LIN {X 104.762,Y 110.384,Z 68.000,A 180.000,B 0.000,C 180.000} C_DIS
LIN {X 105.299,Y 110.068,Z 68.000,A 180.000,B 0.000,C 180.000} C_DIS
LIN {X 105.477,Y 109.954,Z 68.000,A 180.000,B 0.000,C 180.000} C_DIS
LIN {X 105.835,Y 109.715,Z 68.000,A 180.000,B 0.000,C 180.000} C_DIS
LIN {X 106.014,Y 109.595,Z 68.000,A 180.000,B 0.000,C 180.000} C_DIS
LIN {X 106.023,Y 109.589,Z 68.000,A 180.000,B 0.000,C 180.000} C_DIS
LIN {X 106.193,Y 109.465,Z 68.000,A 180.000,B 0.000,C 180.000} C_DIS
LIN {X 106.550,Y 109.196,Z 68.000,A 180.000,B 0.000,C 180.000} C_DIS
LIN {X 106.729,Y 109.060,Z 68.000,A 180.000,B 0.000,C 180.000} C_DIS
LIN {X 106.737,Y 109.053,Z 68.000,A 180.000,B 0.000,C 180.000} C_DIS
LIN {X 106.908,Y 108.910,Z 68.000,A 180.000,B 0.000,C 180.000} C_DIS
LIN {X 107.265,Y 108.608,Z 68.000,A 180.000,B 0.000,C 180.000} C_DIS
LIN {X 107.371,Y 108.517,Z 68.000,A 180.000,B 0.000,C 180.000} C_DIS
LIN {X 107.444,Y 108.448,Z 68.000,A 180.000,B 0.000,C 180.000} C_DIS
LIN {X 107.802,Y 108.110,Z 68.000,A 180.000,B 0.000,C 180.000} C_DIS
LIN {X 107.938,Y 107.980,Z 68.000,A 180.000,B 0.000,C 180.000} C_DIS
LIN {X 107.980,Y 107.938,Z 68.000,A 180.000,B 0.000,C 180.000} C_DIS
LIN {X 108.110,Y 107.802,Z 68.000,A 180.000,B 0.000,C 180.000} C_DIS
LIN {X 108.448,Y 107.444,Z 68.000,A 180.000,B 0.000,C 180.000} C_DIS
LIN {X 108.517,Y 107.371,Z 68.000,A 180.000,B 0.000,C 180.000} C_DIS
LIN {X 108.608,Y 107.265,Z 68.000,A 180.000,B 0.000,C 180.000} C_DIS
LIN {X 108.910,Y 106.908,Z 68.000,A 180.000,B 0.000,C 180.000} C_DIS
LIN {X 109.053,Y 106.737,Z 68.000,A 180.000,B 0.000,C 180.000} C_DIS
LIN {X 109.060,Y 106.729,Z 68.000,A 180.000,B 0.000,C 180.000} C_DIS
LIN {X 109.196,Y 106.550,Z 68.000,A 180.000,B 0.000,C 180.000} C_DIS
LIN {X 109.465,Y 106.193,Z 68.000,A 180.000,B 0.000,C 180.000} C_DIS
LIN {X 109.589,Y 106.023,Z 68.000,A 180.000,B 0.000,C 180.000} C_DIS
LIN {X 109.595,Y 106.014,Z 68.000,A 180.000,B 0.000,C 180.000} C_DIS
LIN {X 109.715,Y 105.835,Z 68.000,A 180.000,B 0.000,C 180.000} C_DIS
LIN {X 109.954,Y 105.477,Z 68.000,A 180.000,B 0.000,C 180.000} C_DIS
LIN {X 110.068,Y 105.299,Z 68.000,A 180.000,B 0.000,C 180.000} C_DIS
LIN {X 110.384,Y 104.762,Z 68.000,A 180.000,B 0.000,C 180.000} C_DIS
LIN {X 110.483,Y 104.586,Z 68.000,A 180.000,B 0.000,C 180.000} C_DIS
LIN {X 110.761,Y 104.047,Z 68.000,A 180.000,B 0.000,C 180.000} C_DIS
LIN {X 110.841,Y 103.889,Z 68.000,A 180.000,B 0.000,C 180.000} C_DIS
LIN {X 110.850,Y 103.869,Z 68.000,A 180.000,B 0.000,C 180.000} C_DIS
LIN {X 110.930,Y 103.690,Z 68.000,A 180.000,B 0.000,C 180.000} C_DIS
LIN {X 111.090,Y 103.332,Z 68.000,A 180.000,B 0.000,C 180.000} C_DIS
LIN {X 111.169,Y 103.153,Z 68.000,A 180.000,B 0.000,C 180.000} C_DIS
LIN {X 111.198,Y 103.079,Z 68.000,A 180.000,B 0.000,C 180.000} C_DIS
LIN {X 111.377,Y 102.610,Z 68.000,A 180.000,B 0.000,C 180.000} C_DIS
LIN {X 111.442,Y 102.438,Z 68.000,A 180.000,B 0.000,C 180.000} C_DIS
LIN {X 111.503,Y 102.260,Z 68.000,A 180.000,B 0.000,C 180.000} C_DIS
LIN {X 111.674,Y 101.723,Z 68.000,A 180.000,B 0.000,C 180.000} C_DIS
LIN {X 111.728,Y 101.545,Z 68.000,A 180.000,B 0.000,C 180.000} C_DIS
LIN {X 111.734,Y 101.518,Z 68.000,A 180.000,B 0.000,C 180.000} C_DIS
LIN {X 111.866,Y 101.008,Z 68.000,A 180.000,B 0.000,C 180.000} C_DIS
LIN {X 111.912,Y 100.829,Z 68.000,A 180.000,B 0.000,C 180.000} C_DIS
LIN {X 111.913,Y 100.824,Z 68.000,A 180.000,B 0.000,C 180.000} C_DIS
LIN {X 111.950,Y 100.651,Z 68.000,A 180.000,B 0.000,C 180.000} C_DIS
LIN {X 112.057,Y 100.114,Z 68.000,A 180.000,B 0.000,C 180.000} C_DIS
LIN {X 112.090,Y 99.936,Z 68.000,A 180.000,B 0.000,C 180.000} C_DIS
LIN {X 112.092,Y 99.919,Z 68.000,A 180.000,B 0.000,C 180.000} C_DIS
LIN {X 112.115,Y 99.757,Z 68.000,A 180.000,B 0.000,C 180.000} C_DIS
LIN {X 112.165,Y 99.399,Z 68.000,A 180.000,B 0.000,C 180.000} C_DIS
LIN {X 112.191,Y 99.221,Z 68.000,A 180.000,B 0.000,C 180.000} C_DIS
LIN {X 112.209,Y 99.042,Z 68.000,A 180.000,B 0.000,C 180.000} C_DIS
LIN {X 112.255,Y 98.505,Z 68.000,A 180.000,B 0.000,C 180.000} C_DIS
LIN {X 112.269,Y 98.327,Z 68.000,A 180.000,B 0.000,C 180.000} C_DIS
LIN {X 112.271,Y 98.281,Z 68.000,A 180.000,B 0.000,C 180.000} C_DIS
LIN {X 112.275,Y 98.148,Z 68.000,A 180.000,B 0.000,C 180.000} C_DIS
LIN {X 112.290,Y 97.612,Z 68.000,A 180.000,B 0.000,C 180.000} C_DIS
LIN {X 112.291,Y 97.433,Z 68.000,A 180.000,B 0.000,C 180.000} C_DIS
LIN {X 112.281,Y 97.075,Z 68.000,A 180.000,B 0.000,C 180.000} C_DIS
LIN {X 112.276,Y 96.897,Z 68.000,A 180.000,B 0.000,C 180.000} C_DIS
LIN {X 112.271,Y 96.719,Z 68.000,A 180.000,B 0.000,C 180.000} C_DIS
LIN {X 112.271,Y 96.718,Z 68.000,A 180.000,B 0.000,C 180.000} C_DIS
LIN {X 112.258,Y 96.539,Z 68.000,A 180.000,B 0.000,C 180.000} C_DIS
LIN {X 112.213,Y 96.003,Z 68.000,A 180.000,B 0.000,C 180.000} C_DIS
LIN {X 112.196,Y 95.824,Z 68.000,A 180.000,B 0.000,C 180.000} C_DIS
LIN {X 112.172,Y 95.645,Z 68.000,A 180.000,B 0.000,C 180.000} C_DIS
LIN {X 112.096,Y 95.109,Z 68.000,A 180.000,B 0.000,C 180.000} C_DIS
LIN {X 112.092,Y 95.081,Z 68.000,A 180.000,B 0.000,C 180.000} C_DIS
LIN {X 112.065,Y 94.930,Z 68.000,A 180.000,B 0.000,C 180.000} C_DIS
LIN {X 111.959,Y 94.394,Z 68.000,A 180.000,B 0.000,C 180.000} C_DIS
LIN {X 111.922,Y 94.215,Z 68.000,A 180.000,B 0.000,C 180.000} C_DIS
LIN {X 111.913,Y 94.176,Z 68.000,A 180.000,B 0.000,C 180.000} C_DIS
LIN {X 111.877,Y 94.036,Z 68.000,A 180.000,B 0.000,C 180.000} C_DIS
LIN {X 111.734,Y 93.482,Z 68.000,A 180.000,B 0.000,C 180.000} C_DIS
LIN {X 111.688,Y 93.321,Z 68.000,A 180.000,B 0.000,C 180.000} C_DIS
LIN {X 111.517,Y 92.785,Z 68.000,A 180.000,B 0.000,C 180.000} C_DIS
LIN {X 111.459,Y 92.606,Z 68.000,A 180.000,B 0.000,C 180.000} C_DIS
LIN {X 111.391,Y 92.427,Z 68.000,A 180.000,B 0.000,C 180.000} C_DIS
LIN {X 111.198,Y 91.921,Z 68.000,A 180.000,B 0.000,C 180.000} C_DIS
LIN {X 111.186,Y 91.891,Z 68.000,A 180.000,B 0.000,C 180.000} C_DIS
LIN {X 111.110,Y 91.712,Z 68.000,A 180.000,B 0.000,C 180.000} C_DIS
LIN {X 110.870,Y 91.176,Z 68.000,A 180.000,B 0.000,C 180.000} C_DIS
LIN {X 110.841,Y 91.111,Z 68.000,A 180.000,B 0.000,C 180.000} C_DIS
LIN {X 110.784,Y 90.997,Z 68.000,A 180.000,B 0.000,C 180.000} C_DIS
LIN {X 110.483,Y 90.414,Z 68.000,A 180.000,B 0.000,C 180.000} C_DIS
LIN {X 110.410,Y 90.282,Z 68.000,A 180.000,B 0.000,C 180.000} C_DIS
LIN {X 110.113,Y 89.778,Z 68.000,A 180.000,B 0.000,C 180.000} C_DIS
; Link Move Starts
LIN {X 109.952,Y 89.519,Z 68.000,A 180.000,B 0.000,C 180.000} C_DIS
LIN {X 109.779,Y 89.258,Z 67.999,A 180.000,B 0.000,C 180.000} C_DIS
LIN {X 109.604,Y 88.996,Z 67.998,A 180.000,B 0.000,C 180.000} C_DIS
LIN {X 109.425,Y 88.751,Z 67.996,A 180.000,B 0.000,C 180.000} C_DIS
LIN {X 109.237,Y 88.499,Z 67.994,A 180.000,B 0.000,C 180.000} C_DIS
LIN {X 109.053,Y 88.256,Z 67.992,A 180.000,B 0.000,C 180.000} C_DIS
LIN {X 108.852,Y 88.015,Z 67.989,A 180.000,B 0.000,C 180.000} C_DIS
LIN {X 108.650,Y 87.773,Z 67.985,A 180.000,B 0.000,C 180.000} C_DIS
LIN {X 108.450,Y 87.544,Z 67.982,A 180.000,B 0.000,C 180.000} C_DIS
LIN {X 108.235,Y 87.314,Z 67.977,A 180.000,B 0.000,C 180.000} C_DIS
LIN {X 108.020,Y 87.084,Z 67.973,A 180.000,B 0.000,C 180.000} C_DIS
LIN {X 107.803,Y 86.870,Z 67.968,A 180.000,B 0.000,C 180.000} C_DIS
LIN {X 107.690,Y 86.761,Z 67.965,A 180.000,B 0.000,C 180.000} C_DIS
LIN {X 107.576,Y 86.652,Z 67.962,A 180.000,B 0.000,C 180.000} C_DIS
LIN {X 107.465,Y 86.545,Z 67.960,A 180.000,B 0.000,C 180.000} C_DIS
LIN {X 107.352,Y 86.439,Z 67.957,A 180.000,B 0.000,C 180.000} C_DIS
LIN {X 107.235,Y 86.338,Z 67.954,A 180.000,B 0.000,C 180.000} C_DIS
LIN {X 107.117,Y 86.236,Z 67.951,A 180.000,B 0.000,C 180.000} C_DIS
LIN {X 106.998,Y 86.134,Z 67.947,A 180.000,B 0.000,C 180.000} C_DIS
LIN {X 106.878,Y 86.031,Z 67.944,A 180.000,B 0.000,C 180.000} C_DIS
LIN {X 106.762,Y 85.931,Z 67.941,A 180.000,B 0.000,C 180.000} C_DIS
LIN {X 106.641,Y 85.835,Z 67.937,A 180.000,B 0.000,C 180.000} C_DIS
LIN {X 106.517,Y 85.740,Z 67.934,A 180.000,B 0.000,C 180.000} C_DIS
LIN {X 106.393,Y 85.645,Z 67.930,A 180.000,B 0.000,C 180.000} C_DIS
LIN {X 106.269,Y 85.549,Z 67.926,A 180.000,B 0.000,C 180.000} C_DIS
LIN {X 106.144,Y 85.453,Z 67.923,A 180.000,B 0.000,C 180.000} C_DIS
LIN {X 106.021,Y 85.363,Z 67.919,A 180.000,B 0.000,C 180.000} C_DIS
LIN {X 105.894,Y 85.276,Z 67.915,A 180.000,B 0.000,C 180.000} C_DIS
LIN {X 105.765,Y 85.187,Z 67.911,A 180.000,B 0.000,C 180.000} C_DIS
LIN {X 105.635,Y 85.098,Z 67.907,A 180.000,B 0.000,C 180.000} C_DIS
LIN {X 105.508,Y 85.011,Z 67.903,A 180.000,B 0.000,C 180.000} C_DIS
LIN {X 105.380,Y 84.926,Z 67.899,A 180.000,B 0.000,C 180.000} C_DIS
LIN {X 105.247,Y 84.844,Z 67.894,A 180.000,B 0.000,C 180.000} C_DIS
LIN {X 105.113,Y 84.762,Z 67.890,A 180.000,B 0.000,C 180.000} C_DIS
LIN {X 104.978,Y 84.680,Z 67.885,A 180.000,B 0.000,C 180.000} C_DIS
LIN {X 104.844,Y 84.599,Z 67.881,A 180.000,B 0.000,C 180.000} C_DIS
LIN {X 104.712,Y 84.519,Z 67.876,A 180.000,B 0.000,C 180.000} C_DIS
LIN {X 104.577,Y 84.444,Z 67.872,A 180.000,B 0.000,C 180.000} C_DIS
LIN {X 104.439,Y 84.370,Z 67.867,A 180.000,B 0.000,C 180.000} C_DIS
LIN {X 104.300,Y 84.296,Z 67.862,A 180.000,B 0.000,C 180.000} C_DIS
LIN {X 104.162,Y 84.222,Z 67.857,A 180.000,B 0.000,C 180.000} C_DIS
LIN {X 104.023,Y 84.148,Z 67.852,A 180.000,B 0.000,C 180.000} C_DIS
LIN {X 103.885,Y 84.079,Z 67.847,A 180.000,B 0.000,C 180.000} C_DIS
LIN {X 103.746,Y 84.014,Z 67.842,A 180.000,B 0.000,C 180.000} C_DIS
LIN {X 103.675,Y 83.981,Z 67.840,A 180.000,B 0.000,C 180.000} C_DIS
LIN {X 103.603,Y 83.947,Z 67.837,A 180.000,B 0.000,C 180.000} C_DIS
LIN {X 103.532,Y 83.914,Z 67.835,A 180.000,B 0.000,C 180.000} C_DIS
LIN {X 103.390,Y 83.848,Z 67.829,A 180.000,B 0.000,C 180.000} C_DIS
LIN {X 103.319,Y 83.815,Z 67.827,A 180.000,B 0.000,C 180.000} C_DIS
LIN {X 103.249,Y 83.782,Z 67.824,A 180.000,B 0.000,C 180.000} C_DIS
LIN {X 103.178,Y 83.751,Z 67.821,A 180.000,B 0.000,C 180.000} C_DIS
LIN {X 103.106,Y 83.721,Z 67.819,A 180.000,B 0.000,C 180.000} C_DIS
LIN {X 103.033,Y 83.692,Z 67.816,A 180.000,B 0.000,C 180.000} C_DIS
LIN {X 102.888,Y 83.634,Z 67.811,A 180.000,B 0.000,C 180.000} C_DIS
LIN {X 102.742,Y 83.576,Z 67.805,A 180.000,B 0.000,C 180.000} C_DIS
LIN {X 102.524,Y 83.488,Z 67.797,A 180.000,B 0.000,C 180.000} C_DIS
LIN {X 102.453,Y 83.460,Z 67.794,A 180.000,B 0.000,C 180.000} C_DIS
LIN {X 102.380,Y 83.433,Z 67.792,A 180.000,B 0.000,C 180.000} C_DIS
LIN {X 102.307,Y 83.408,Z 67.789,A 180.000,B 0.000,C 180.000} C_DIS
LIN {X 102.158,Y 83.358,Z 67.783,A 180.000,B 0.000,C 180.000} C_DIS
LIN {X 101.934,Y 83.283,Z 67.775,A 180.000,B 0.000,C 180.000} C_DIS
LIN {X 101.784,Y 83.232,Z 67.770,A 180.000,B 0.000,C 180.000} C_DIS
LIN {X 101.710,Y 83.207,Z 67.767,A 180.000,B 0.000,C 180.000} C_DIS
LIN {X 101.636,Y 83.183,Z 67.764,A 180.000,B 0.000,C 180.000} C_DIS
LIN {X 101.562,Y 83.161,Z 67.762,A 180.000,B 0.000,C 180.000} C_DIS
LIN {X 101.413,Y 83.120,Z 67.756,A 180.000,B 0.000,C 180.000} C_DIS
LIN {X 101.261,Y 83.078,Z 67.751,A 180.000,B 0.000,C 180.000} C_DIS
LIN {X 101.034,Y 83.016,Z 67.742,A 180.000,B 0.000,C 180.000} C_DIS
LIN {X 100.884,Y 82.975,Z 67.737,A 180.000,B 0.000,C 180.000} C_DIS
LIN {X 100.809,Y 82.955,Z 67.734,A 180.000,B 0.000,C 180.000} C_DIS
LIN {X 100.732,Y 82.938,Z 67.732,A 180.000,B 0.000,C 180.000} C_DIS
LIN {X 100.578,Y 82.905,Z 67.726,A 180.000,B 0.000,C 180.000} C_DIS
LIN {X 100.502,Y 82.888,Z 67.723,A 180.000,B 0.000,C 180.000} C_DIS
LIN {X 100.348,Y 82.855,Z 67.718,A 180.000,B 0.000,C 180.000} C_DIS
LIN {X 100.118,Y 82.805,Z 67.710,A 180.000,B 0.000,C 180.000} C_DIS
LIN {X 100.042,Y 82.789,Z 67.707,A 180.000,B 0.000,C 180.000} C_DIS
LIN {X 99.965,Y 82.775,Z 67.704,A 180.000,B 0.000,C 180.000} C_DIS
LIN {X 99.888,Y 82.762,Z 67.701,A 180.000,B 0.000,C 180.000} C_DIS
LIN {X 99.733,Y 82.738,Z 67.696,A 180.000,B 0.000,C 180.000} C_DIS
LIN {X 99.266,Y 82.664,Z 67.679,A 180.000,B 0.000,C 180.000} C_DIS
LIN {X 99.189,Y 82.653,Z 67.677,A 180.000,B 0.000,C 180.000} C_DIS
LIN {X 99.112,Y 82.643,Z 67.674,A 180.000,B 0.000,C 180.000} C_DIS
LIN {X 98.956,Y 82.628,Z 67.669,A 180.000,B 0.000,C 180.000} C_DIS
LIN {X 98.800,Y 82.612,Z 67.663,A 180.000,B 0.000,C 180.000} C_DIS
LIN {X 98.408,Y 82.572,Z 67.649,A 180.000,B 0.000,C 180.000} C_DIS
LIN {X 98.330,Y 82.566,Z 67.647,A 180.000,B 0.000,C 180.000} C_DIS
LIN {X 98.252,Y 82.562,Z 67.644,A 180.000,B 0.000,C 180.000} C_DIS
LIN {X 97.781,Y 82.541,Z 67.627,A 180.000,B 0.000,C 180.000} C_DIS
LIN {X 97.624,Y 82.534,Z 67.622,A 180.000,B 0.000,C 180.000} C_DIS
LIN {X 97.546,Y 82.530,Z 67.619,A 180.000,B 0.000,C 180.000} C_DIS
LIN {X 97.467,Y 82.529,Z 67.616,A 180.000,B 0.000,C 180.000} C_DIS
LIN {X 97.389,Y 82.530,Z 67.614,A 180.000,B 0.000,C 180.000} C_DIS
LIN {X 97.153,Y 82.532,Z 67.605,A 180.000,B 0.000,C 180.000} C_DIS
LIN {X 96.995,Y 82.534,Z 67.600,A 180.000,B 0.000,C 180.000} C_DIS
LIN {X 96.759,Y 82.537,Z 67.592,A 180.000,B 0.000,C 180.000} C_DIS
LIN {X 96.680,Y 82.538,Z 67.589,A 180.000,B 0.000,C 180.000} C_DIS
LIN {X 96.602,Y 82.542,Z 67.586,A 180.000,B 0.000,C 180.000} C_DIS
LIN {X 96.524,Y 82.547,Z 67.583,A 180.000,B 0.000,C 180.000} C_DIS
LIN {X 96.131,Y 82.574,Z 67.570,A 180.000,B 0.000,C 180.000} C_DIS
LIN {X 95.895,Y 82.590,Z 67.561,A 180.000,B 0.000,C 180.000} C_DIS
LIN {X 95.817,Y 82.597,Z 67.559,A 180.000,B 0.000,C 180.000} C_DIS
LIN {X 95.739,Y 82.605,Z 67.556,A 180.000,B 0.000,C 180.000} C_DIS
LIN {X 95.709,Y 82.609,Z 67.555,A 180.000,B 0.000,C 180.000} C_DIS
LIN {X 95.115,Y 82.693,Z 67.534,A 180.000,B 0.000,C 180.000} C_DIS
LIN {X 95.037,Y 82.704,Z 67.531,A 180.000,B 0.000,C 180.000} C_DIS
LIN {X 94.959,Y 82.717,Z 67.528,A 180.000,B 0.000,C 180.000} C_DIS
LIN {X 94.882,Y 82.732,Z 67.526,A 180.000,B 0.000,C 180.000} C_DIS
LIN {X 94.264,Y 82.855,Z 67.504,A 180.000,B 0.000,C 180.000} C_DIS
LIN {X 94.187,Y 82.871,Z 67.501,A 180.000,B 0.000,C 180.000} C_DIS
LIN {X 94.110,Y 82.889,Z 67.498,A 180.000,B 0.000,C 180.000} C_DIS
LIN {X 94.034,Y 82.908,Z 67.495,A 180.000,B 0.000,C 180.000} C_DIS
LIN {X 93.424,Y 83.066,Z 67.473,A 180.000,B 0.000,C 180.000} C_DIS
LIN {X 93.348,Y 83.086,Z 67.471,A 180.000,B 0.000,C 180.000} C_DIS
LIN {X 93.272,Y 83.109,Z 67.468,A 180.000,B 0.000,C 180.000} C_DIS
LIN {X 92.672,Y 83.300,Z 67.446,A 180.000,B 0.000,C 180.000} C_DIS
LIN {X 92.597,Y 83.324,Z 67.443,A 180.000,B 0.000,C 180.000} C_DIS
LIN {X 92.523,Y 83.350,Z 67.440,A 180.000,B 0.000,C 180.000} C_DIS
LIN {X 92.449,Y 83.378,Z 67.438,A 180.000,B 0.000,C 180.000} C_DIS
LIN {X 92.007,Y 83.546,Z 67.421,A 180.000,B 0.000,C 180.000} C_DIS
LIN {X 91.860,Y 83.602,Z 67.416,A 180.000,B 0.000,C 180.000} C_DIS
LIN {X 91.787,Y 83.631,Z 67.413,A 180.000,B 0.000,C 180.000} C_DIS
LIN {X 91.714,Y 83.661,Z 67.410,A 180.000,B 0.000,C 180.000} C_DIS
LIN {X 91.642,Y 83.693,Z 67.407,A 180.000,B 0.000,C 180.000} C_DIS
LIN {X 91.427,Y 83.790,Z 67.399,A 180.000,B 0.000,C 180.000} C_DIS
LIN {X 91.067,Y 83.951,Z 67.385,A 180.000,B 0.000,C 180.000} C_DIS
LIN {X 90.996,Y 83.984,Z 67.383,A 180.000,B 0.000,C 180.000} C_DIS
LIN {X 90.925,Y 84.019,Z 67.380,A 180.000,B 0.000,C 180.000} C_DIS
LIN {X 90.505,Y 84.236,Z 67.363,A 180.000,B 0.000,C 180.000} C_DIS
LIN {X 90.365,Y 84.308,Z 67.358,A 180.000,B 0.000,C 180.000} C_DIS
LIN {X 90.296,Y 84.344,Z 67.355,A 180.000,B 0.000,C 180.000} C_DIS
LIN {X 90.226,Y 84.382,Z 67.352,A 180.000,B 0.000,C 180.000} C_DIS
LIN {X 90.158,Y 84.421,Z 67.350,A 180.000,B 0.000,C 180.000} C_DIS
LIN {X 89.955,Y 84.541,Z 67.341,A 180.000,B 0.000,C 180.000} C_DIS
LIN {X 89.819,Y 84.621,Z 67.336,A 180.000,B 0.000,C 180.000} C_DIS
LIN {X 89.683,Y 84.701,Z 67.330,A 180.000,B 0.000,C 180.000} C_DIS
LIN {X 89.616,Y 84.741,Z 67.328,A 180.000,B 0.000,C 180.000} C_DIS
LIN {X 89.548,Y 84.782,Z 67.325,A 180.000,B 0.000,C 180.000} C_DIS
LIN {X 89.481,Y 84.824,Z 67.322,A 180.000,B 0.000,C 180.000} C_DIS
LIN {X 89.416,Y 84.867,Z 67.319,A 180.000,B 0.000,C 180.000} C_DIS
LIN {X 89.350,Y 84.911,Z 67.317,A 180.000,B 0.000,C 180.000} C_DIS
LIN {X 89.219,Y 84.999,Z 67.311,A 180.000,B 0.000,C 180.000} C_DIS
LIN {X 88.892,Y 85.217,Z 67.297,A 180.000,B 0.000,C 180.000} C_DIS
LIN {X 88.827,Y 85.262,Z 67.295,A 180.000,B 0.000,C 180.000} C_DIS
LIN {X 88.763,Y 85.308,Z 67.292,A 180.000,B 0.000,C 180.000} C_DIS
LIN {X 88.637,Y 85.403,Z 67.286,A 180.000,B 0.000,C 180.000} C_DIS
LIN {X 88.574,Y 85.450,Z 67.284,A 180.000,B 0.000,C 180.000} C_DIS
LIN {X 88.449,Y 85.545,Z 67.278,A 180.000,B 0.000,C 180.000} C_DIS
LIN {X 88.260,Y 85.687,Z 67.270,A 180.000,B 0.000,C 180.000} C_DIS
LIN {X 88.197,Y 85.734,Z 67.267,A 180.000,B 0.000,C 180.000} C_DIS
LIN {X 88.135,Y 85.783,Z 67.265,A 180.000,B 0.000,C 180.000} C_DIS
LIN {X 88.074,Y 85.833,Z 67.262,A 180.000,B 0.000,C 180.000} C_DIS
LIN {X 87.954,Y 85.935,Z 67.256,A 180.000,B 0.000,C 180.000} C_DIS
LIN {X 87.774,Y 86.087,Z 67.248,A 180.000,B 0.000,C 180.000} C_DIS
LIN {X 87.653,Y 86.189,Z 67.243,A 180.000,B 0.000,C 180.000} C_DIS
LIN {X 87.593,Y 86.240,Z 67.240,A 180.000,B 0.000,C 180.000} C_DIS
LIN {X 87.533,Y 86.291,Z 67.237,A 180.000,B 0.000,C 180.000} C_DIS
LIN {X 87.474,Y 86.343,Z 67.234,A 180.000,B 0.000,C 180.000} C_DIS
LIN {X 87.417,Y 86.397,Z 67.232,A 180.000,B 0.000,C 180.000} C_DIS
LIN {X 87.360,Y 86.451,Z 67.229,A 180.000,B 0.000,C 180.000} C_DIS
LIN {X 87.245,Y 86.559,Z 67.223,A 180.000,B 0.000,C 180.000} C_DIS
LIN {X 87.074,Y 86.722,Z 67.215,A 180.000,B 0.000,C 180.000} C_DIS
LIN {X 86.959,Y 86.830,Z 67.210,A 180.000,B 0.000,C 180.000} C_DIS
LIN {X 86.902,Y 86.884,Z 67.207,A 180.000,B 0.000,C 180.000} C_DIS
LIN {X 86.847,Y 86.941,Z 67.204,A 180.000,B 0.000,C 180.000} C_DIS
LIN {X 86.739,Y 87.055,Z 67.199,A 180.000,B 0.000,C 180.000} C_DIS
LIN {X 86.685,Y 87.112,Z 67.196,A 180.000,B 0.000,C 180.000} C_DIS
LIN {X 86.577,Y 87.227,Z 67.190,A 180.000,B 0.000,C 180.000} C_DIS
LIN {X 86.469,Y 87.341,Z 67.185,A 180.000,B 0.000,C 180.000} C_DIS
LIN {X 86.360,Y 87.456,Z 67.179,A 180.000,B 0.000,C 180.000} C_DIS
LIN {X 86.307,Y 87.514,Z 67.177,A 180.000,B 0.000,C 180.000} C_DIS
LIN {X 86.256,Y 87.574,Z 67.174,A 180.000,B 0.000,C 180.000} C_DIS
LIN {X 86.154,Y 87.694,Z 67.169,A 180.000,B 0.000,C 180.000} C_DIS
LIN {X 86.053,Y 87.814,Z 67.164,A 180.000,B 0.000,C 180.000} C_DIS
LIN {X 86.002,Y 87.874,Z 67.161,A 180.000,B 0.000,C 180.000} C_DIS
LIN {X 85.951,Y 87.935,Z 67.158,A 180.000,B 0.000,C 180.000} C_DIS
LIN {X 85.900,Y 87.995,Z 67.156,A 180.000,B 0.000,C 180.000} C_DIS
LIN {X 85.850,Y 88.055,Z 67.153,A 180.000,B 0.000,C 180.000} C_DIS
LIN {X 85.799,Y 88.115,Z 67.151,A 180.000,B 0.000,C 180.000} C_DIS
LIN {X 85.750,Y 88.177,Z 67.148,A 180.000,B 0.000,C 180.000} C_DIS
LIN {X 85.655,Y 88.302,Z 67.143,A 180.000,B 0.000,C 180.000} C_DIS
LIN {X 85.560,Y 88.428,Z 67.138,A 180.000,B 0.000,C 180.000} C_DIS
LIN {X 85.465,Y 88.554,Z 67.134,A 180.000,B 0.000,C 180.000} C_DIS
LIN {X 85.371,Y 88.680,Z 67.129,A 180.000,B 0.000,C 180.000} C_DIS
LIN {X 85.276,Y 88.806,Z 67.124,A 180.000,B 0.000,C 180.000} C_DIS
LIN {X 85.188,Y 88.936,Z 67.120,A 180.000,B 0.000,C 180.000} C_DIS
LIN {X 85.100,Y 89.067,Z 67.115,A 180.000,B 0.000,C 180.000} C_DIS
LIN {X 85.013,Y 89.198,Z 67.110,A 180.000,B 0.000,C 180.000} C_DIS
LIN {X 84.925,Y 89.329,Z 67.106,A 180.000,B 0.000,C 180.000} C_DIS
LIN {X 84.838,Y 89.460,Z 67.102,A 180.000,B 0.000,C 180.000} C_DIS
LIN {X 84.754,Y 89.594,Z 67.097,A 180.000,B 0.000,C 180.000} C_DIS
LIN {X 84.674,Y 89.729,Z 67.093,A 180.000,B 0.000,C 180.000} C_DIS
LIN {X 84.594,Y 89.865,Z 67.089,A 180.000,B 0.000,C 180.000} C_DIS
LIN {X 84.514,Y 90.001,Z 67.085,A 180.000,B 0.000,C 180.000} C_DIS
LIN {X 84.434,Y 90.136,Z 67.081,A 180.000,B 0.000,C 180.000} C_DIS
LIN {X 84.356,Y 90.273,Z 67.077,A 180.000,B 0.000,C 180.000} C_DIS
LIN {X 84.283,Y 90.413,Z 67.073,A 180.000,B 0.000,C 180.000} C_DIS
LIN {X 84.211,Y 90.553,Z 67.070,A 180.000,B 0.000,C 180.000} C_DIS
LIN {X 84.139,Y 90.693,Z 67.066,A 180.000,B 0.000,C 180.000} C_DIS
LIN {X 84.067,Y 90.833,Z 67.062,A 180.000,B 0.000,C 180.000} C_DIS
LIN {X 83.995,Y 90.973,Z 67.059,A 180.000,B 0.000,C 180.000} C_DIS
LIN {X 83.929,Y 91.116,Z 67.056,A 180.000,B 0.000,C 180.000} C_DIS
LIN {X 83.865,Y 91.260,Z 67.052,A 180.000,B 0.000,C 180.000} C_DIS
LIN {X 83.800,Y 91.403,Z 67.049,A 180.000,B 0.000,C 180.000} C_DIS
LIN {X 83.736,Y 91.547,Z 67.046,A 180.000,B 0.000,C 180.000} C_DIS
LIN {X 83.672,Y 91.691,Z 67.043,A 180.000,B 0.000,C 180.000} C_DIS
LIN {X 83.611,Y 91.837,Z 67.040,A 180.000,B 0.000,C 180.000} C_DIS
LIN {X 83.555,Y 91.984,Z 67.037,A 180.000,B 0.000,C 180.000} C_DIS
LIN {X 83.499,Y 92.131,Z 67.034,A 180.000,B 0.000,C 180.000} C_DIS
LIN {X 83.443,Y 92.278,Z 67.032,A 180.000,B 0.000,C 180.000} C_DIS
LIN {X 83.387,Y 92.425,Z 67.029,A 180.000,B 0.000,C 180.000} C_DIS
LIN {X 83.284,Y 92.723,Z 67.024,A 180.000,B 0.000,C 180.000} C_DIS
LIN {X 83.189,Y 93.023,Z 67.020,A 180.000,B 0.000,C 180.000} C_DIS
LIN {X 83.093,Y 93.323,Z 67.016,A 180.000,B 0.000,C 180.000} C_DIS
LIN {X 83.013,Y 93.628,Z 67.013,A 180.000,B 0.000,C 180.000} C_DIS
LIN {X 82.934,Y 93.933,Z 67.009,A 180.000,B 0.000,C 180.000} C_DIS
LIN {X 82.860,Y 94.239,Z 67.007,A 180.000,B 0.000,C 180.000} C_DIS
LIN {X 82.798,Y 94.548,Z 67.004,A 180.000,B 0.000,C 180.000} C_DIS
LIN {X 82.737,Y 94.857,Z 67.003,A 180.000,B 0.000,C 180.000} C_DIS
LIN {X 82.686,Y 95.167,Z 67.001,A 180.000,B 0.000,C 180.000} C_DIS
LIN {X 82.641,Y 95.479,Z 67.000,A 180.000,B 0.000,C 180.000} C_DIS
LIN {X 82.598,Y 95.791,Z 67.000,A 180.000,B 0.000,C 180.000} C_DIS
LIN {X 82.589,Y 95.875,Z 67.000,A 180.000,B 0.000,C 180.000} C_DIS
; Cutting Move Starts
LIN {X 82.578,Y 96.003,Z 67.000,A 180.000,B 0.000,C 180.000} C_DIS
LIN {X 82.533,Y 96.539,Z 67.000,A 180.000,B 0.000,C 180.000} C_DIS
LIN {X 82.521,Y 96.718,Z 67.000,A 180.000,B 0.000,C 180.000} C_DIS
LIN {X 82.516,Y 96.897,Z 67.000,A 180.000,B 0.000,C 180.000} C_DIS
LIN {X 82.501,Y 97.433,Z 67.000,A 180.000,B 0.000,C 180.000} C_DIS
LIN {X 82.502,Y 97.612,Z 67.000,A 180.000,B 0.000,C 180.000} C_DIS
LIN {X 82.517,Y 98.148,Z 67.000,A 180.000,B 0.000,C 180.000} C_DIS
LIN {X 82.523,Y 98.327,Z 67.000,A 180.000,B 0.000,C 180.000} C_DIS
LIN {X 82.536,Y 98.505,Z 67.000,A 180.000,B 0.000,C 180.000} C_DIS
LIN {X 82.582,Y 99.042,Z 67.000,A 180.000,B 0.000,C 180.000} C_DIS
LIN {X 82.595,Y 99.185,Z 67.000,A 180.000,B 0.000,C 180.000} C_DIS
LIN {X 82.599,Y 99.221,Z 67.000,A 180.000,B 0.000,C 180.000} C_DIS
LIN {X 82.624,Y 99.399,Z 67.000,A 180.000,B 0.000,C 180.000} C_DIS
LIN {X 82.700,Y 99.936,Z 67.000,A 180.000,B 0.000,C 180.000} C_DIS
LIN {X 82.731,Y 100.114,Z 67.000,A 180.000,B 0.000,C 180.000} C_DIS
LIN {X 82.838,Y 100.651,Z 67.000,A 180.000,B 0.000,C 180.000} C_DIS
LIN {X 82.874,Y 100.829,Z 67.000,A 180.000,B 0.000,C 180.000} C_DIS
LIN {X 82.919,Y 101.008,Z 67.000,A 180.000,B 0.000,C 180.000} C_DIS
LIN {X 83.057,Y 101.545,Z 67.000,A 180.000,B 0.000,C 180.000} C_DIS
LIN {X 83.108,Y 101.723,Z 67.000,A 180.000,B 0.000,C 180.000} C_DIS
LIN {X 83.310,Y 102.358,Z 67.000,A 180.000,B 0.000,C 180.000} C_DIS
LIN {X 83.336,Y 102.438,Z 67.000,A 180.000,B 0.000,C 180.000} C_DIS
LIN {X 83.403,Y 102.617,Z 67.000,A 180.000,B 0.000,C 180.000} C_DIS
LIN {X 83.608,Y 103.153,Z 67.000,A 180.000,B 0.000,C 180.000} C_DIS
LIN {X 83.668,Y 103.300,Z 67.000,A 180.000,B 0.000,C 180.000} C_DIS
LIN {X 83.922,Y 103.869,Z 67.000,A 180.000,B 0.000,C 180.000} C_DIS
LIN {X 84.005,Y 104.047,Z 67.000,A 180.000,B 0.000,C 180.000} C_DIS
LIN {X 84.025,Y 104.087,Z 67.000,A 180.000,B 0.000,C 180.000} C_DIS
LIN {X 84.282,Y 104.584,Z 67.000,A 180.000,B 0.000,C 180.000} C_DIS
LIN {X 84.375,Y 104.762,Z 67.000,A 180.000,B 0.000,C 180.000} C_DIS
LIN {X 84.383,Y 104.775,Z 67.000,A 180.000,B 0.000,C 180.000} C_DIS
LIN {X 84.480,Y 104.941,Z 67.000,A 180.000,B 0.000,C 180.000} C_DIS
LIN {X 84.740,Y 105.382,Z 67.000,A 180.000,B 0.000,C 180.000} C_DIS
LIN {X 84.797,Y 105.477,Z 67.000,A 180.000,B 0.000,C 180.000} C_DIS
LIN {X 84.915,Y 105.656,Z 67.000,A 180.000,B 0.000,C 180.000} C_DIS
LIN {X 85.154,Y 106.014,Z 67.000,A 180.000,B 0.000,C 180.000} C_DIS
LIN {X 85.276,Y 106.193,Z 67.000,A 180.000,B 0.000,C 180.000} C_DIS
LIN {X 85.276,Y 106.194,Z 67.000,A 180.000,B 0.000,C 180.000} C_DIS
LIN {X 85.409,Y 106.371,Z 67.000,A 180.000,B 0.000,C 180.000} C_DIS
LIN {X 85.678,Y 106.729,Z 67.000,A 180.000,B 0.000,C 180.000} C_DIS
LIN {X 85.813,Y 106.902,Z 67.000,A 180.000,B 0.000,C 180.000} C_DIS
LIN {X 85.818,Y 106.908,Z 67.000,A 180.000,B 0.000,C 180.000} C_DIS
LIN {X 86.271,Y 107.444,Z 67.000,A 180.000,B 0.000,C 180.000} C_DIS
LIN {X 86.349,Y 107.532,Z 67.000,A 180.000,B 0.000,C 180.000} C_DIS
LIN {X 86.435,Y 107.623,Z 67.000,A 180.000,B 0.000,C 180.000} C_DIS
LIN {X 86.773,Y 107.980,Z 67.000,A 180.000,B 0.000,C 180.000} C_DIS
LIN {X 86.885,Y 108.099,Z 67.000,A 180.000,B 0.000,C 180.000} C_DIS
LIN {X 86.947,Y 108.159,Z 67.000,A 180.000,B 0.000,C 180.000} C_DIS
LIN {X 87.422,Y 108.607,Z 67.000,A 180.000,B 0.000,C 180.000} C_DIS
LIN {X 87.517,Y 108.695,Z 67.000,A 180.000,B 0.000,C 180.000} C_DIS
LIN {X 87.601,Y 108.767,Z 67.000,A 180.000,B 0.000,C 180.000} C_DIS
LIN {X 87.958,Y 109.069,Z 67.000,A 180.000,B 0.000,C 180.000} C_DIS
LIN {X 88.137,Y 109.219,Z 67.000,A 180.000,B 0.000,C 180.000} C_DIS
LIN {X 88.153,Y 109.232,Z 67.000,A 180.000,B 0.000,C 180.000} C_DIS
LIN {X 88.316,Y 109.355,Z 67.000,A 180.000,B 0.000,C 180.000} C_DIS
LIN {X 88.673,Y 109.624,Z 67.000,A 180.000,B 0.000,C 180.000} C_DIS
LIN {X 88.852,Y 109.756,Z 67.000,A 180.000,B 0.000,C 180.000} C_DIS
LIN {X 88.870,Y 109.768,Z 67.000,A 180.000,B 0.000,C 180.000} C_DIS
LIN {X 89.031,Y 109.875,Z 67.000,A 180.000,B 0.000,C 180.000} C_DIS
LIN {X 89.405,Y 110.126,Z 67.000,A 180.000,B 0.000,C 180.000} C_DIS
LIN {X 89.567,Y 110.230,Z 67.000,A 180.000,B 0.000,C 180.000} C_DIS
LIN {X 89.693,Y 110.304,Z 67.000,A 180.000,B 0.000,C 180.000} C_DIS
LIN {X 90.103,Y 110.546,Z 67.000,A 180.000,B 0.000,C 180.000} C_DIS
LIN {X 90.282,Y 110.649,Z 67.000,A 180.000,B 0.000,C 180.000} C_DIS
LIN {X 90.307,Y 110.662,Z 67.000,A 180.000,B 0.000,C 180.000} C_DIS
LIN {X 90.818,Y 110.926,Z 67.000,A 180.000,B 0.000,C 180.000} C_DIS
LIN {X 90.997,Y 111.017,Z 67.000,A 180.000,B 0.000,C 180.000} C_DIS
LIN {X 91.002,Y 111.019,Z 67.000,A 180.000,B 0.000,C 180.000} C_DIS
LIN {X 91.176,Y 111.098,Z 67.000,A 180.000,B 0.000,C 180.000} C_DIS
LIN {X 91.533,Y 111.258,Z 67.000,A 180.000,B 0.000,C 180.000} C_DIS
LIN {X 91.712,Y 111.338,Z 67.000,A 180.000,B 0.000,C 180.000} C_DIS
LIN {X 91.806,Y 111.377,Z 67.000,A 180.000,B 0.000,C 180.000} C_DIS
LIN {X 91.891,Y 111.409,Z 67.000,A 180.000,B 0.000,C 180.000} C_DIS
LIN {X 92.427,Y 111.614,Z 67.000,A 180.000,B 0.000,C 180.000} C_DIS
LIN {X 92.606,Y 111.678,Z 67.000,A 180.000,B 0.000,C 180.000} C_DIS
LIN {X 92.964,Y 111.792,Z 67.000,A 180.000,B 0.000,C 180.000} C_DIS
LIN {X 93.142,Y 111.849,Z 67.000,A 180.000,B 0.000,C 180.000} C_DIS
LIN {X 93.321,Y 111.906,Z 67.000,A 180.000,B 0.000,C 180.000} C_DIS
LIN {X 93.346,Y 111.913,Z 67.000,A 180.000,B 0.000,C 180.000} C_DIS
LIN {X 93.500,Y 111.954,Z 67.000,A 180.000,B 0.000,C 180.000} C_DIS
LIN {X 94.036,Y 112.092,Z 67.000,A 180.000,B 0.000,C 180.000} C_DIS
LIN {X 94.215,Y 112.135,Z 67.000,A 180.000,B 0.000,C 180.000} C_DIS
LIN {X 94.394,Y 112.171,Z 67.000,A 180.000,B 0.000,C 180.000} C_DIS
LIN {X 94.895,Y 112.271,Z 67.000,A 180.000,B 0.000,C 180.000} C_DIS
LIN {X 94.930,Y 112.278,Z 67.000,A 180.000,B 0.000,C 180.000} C_DIS
LIN {X 95.109,Y 112.306,Z 67.000,A 180.000,B 0.000,C 180.000} C_DIS
LIN {X 95.645,Y 112.382,Z 67.000,A 180.000,B 0.000,C 180.000} C_DIS
LIN {X 95.824,Y 112.406,Z 67.000,A 180.000,B 0.000,C 180.000} C_DIS
LIN {X 96.003,Y 112.422,Z 67.000,A 180.000,B 0.000,C 180.000} C_DIS
LIN {X 96.539,Y 112.467,Z 67.000,A 180.000,B 0.000,C 180.000} C_DIS
LIN {X 96.718,Y 112.479,Z 67.000,A 180.000,B 0.000,C 180.000} C_DIS
LIN {X 96.897,Y 112.484,Z 67.000,A 180.000,B 0.000,C 180.000} C_DIS
LIN {X 97.433,Y 112.499,Z 67.000,A 180.000,B 0.000,C 180.000} C_DIS
LIN {X 97.612,Y 112.498,Z 67.000,A 180.000,B 0.000,C 180.000} C_DIS
LIN {X 98.148,Y 112.483,Z 67.000,A 180.000,B 0.000,C 180.000} C_DIS
LIN {X 98.327,Y 112.477,Z 67.000,A 180.000,B 0.000,C 180.000} C_DIS
LIN {X 98.505,Y 112.464,Z 67.000,A 180.000,B 0.000,C 180.000} C_DIS
LIN {X 99.042,Y 112.418,Z 67.000,A 180.000,B 0.000,C 180.000} C_DIS
LIN {X 99.221,Y 112.401,Z 67.000,A 180.000,B 0.000,C 180.000} C_DIS
LIN {X 99.399,Y 112.376,Z 67.000,A 180.000,B 0.000,C 180.000} C_DIS
LIN {X 99.936,Y 112.300,Z 67.000,A 180.000,B 0.000,C 180.000} C_DIS
LIN {X 100.105,Y 112.271,Z 67.000,A 180.000,B 0.000,C 180.000} C_DIS
LIN {X 100.651,Y 112.162,Z 67.000,A 180.000,B 0.000,C 180.000} C_DIS
LIN {X 100.829,Y 112.126,Z 67.000,A 180.000,B 0.000,C 180.000} C_DIS
LIN {X 100.966,Y 112.092,Z 67.000,A 180.000,B 0.000,C 180.000} C_DIS
LIN {X 101.545,Y 111.943,Z 67.000,A 180.000,B 0.000,C 180.000} C_DIS
LIN {X 101.654,Y 111.913,Z 67.000,A 180.000,B 0.000,C 180.000} C_DIS
LIN {X 101.723,Y 111.892,Z 67.000,A 180.000,B 0.000,C 180.000} C_DIS
LIN {X 102.260,Y 111.721,Z 67.000,A 180.000,B 0.000,C 180.000} C_DIS
LIN {X 102.438,Y 111.664,Z 67.000,A 180.000,B 0.000,C 180.000} C_DIS
LIN {X 102.617,Y 111.597,Z 67.000,A 180.000,B 0.000,C 180.000} C_DIS
LIN {X 103.153,Y 111.392,Z 67.000,A 180.000,B 0.000,C 180.000} C_DIS
LIN {X 103.194,Y 111.377,Z 67.000,A 180.000,B 0.000,C 180.000} C_DIS
LIN {X 103.332,Y 111.318,Z 67.000,A 180.000,B 0.000,C 180.000} C_DIS
LIN {X 103.869,Y 111.078,Z 67.000,A 180.000,B 0.000,C 180.000} C_DIS
LIN {X 103.998,Y 111.019,Z 67.000,A 180.000,B 0.000,C 180.000} C_DIS
LIN {X 104.047,Y 110.995,Z 67.000,A 180.000,B 0.000,C 180.000} C_DIS
LIN {X 104.226,Y 110.903,Z 67.000,A 180.000,B 0.000,C 180.000} C_DIS
LIN {X 104.693,Y 110.662,Z 67.000,A 180.000,B 0.000,C 180.000} C_DIS
LIN {X 104.762,Y 110.625,Z 67.000,A 180.000,B 0.000,C 180.000} C_DIS
LIN {X 104.941,Y 110.520,Z 67.000,A 180.000,B 0.000,C 180.000} C_DIS
LIN {X 105.307,Y 110.304,Z 67.000,A 180.000,B 0.000,C 180.000} C_DIS
LIN {X 105.477,Y 110.203,Z 67.000,A 180.000,B 0.000,C 180.000} C_DIS
LIN {X 105.595,Y 110.126,Z 67.000,A 180.000,B 0.000,C 180.000} C_DIS
LIN {X 106.014,Y 109.846,Z 67.000,A 180.000,B 0.000,C 180.000} C_DIS
LIN {X 106.130,Y 109.768,Z 67.000,A 180.000,B 0.000,C 180.000} C_DIS
LIN {X 106.193,Y 109.724,Z 67.000,A 180.000,B 0.000,C 180.000} C_DIS
LIN {X 106.371,Y 109.591,Z 67.000,A 180.000,B 0.000,C 180.000} C_DIS
LIN {X 106.729,Y 109.322,Z 67.000,A 180.000,B 0.000,C 180.000} C_DIS
LIN {X 106.847,Y 109.232,Z 67.000,A 180.000,B 0.000,C 180.000} C_DIS
LIN {X 106.908,Y 109.182,Z 67.000,A 180.000,B 0.000,C 180.000} C_DIS
LIN {X 107.444,Y 108.729,Z 67.000,A 180.000,B 0.000,C 180.000} C_DIS
LIN {X 107.483,Y 108.695,Z 67.000,A 180.000,B 0.000,C 180.000} C_DIS
LIN {X 107.623,Y 108.565,Z 67.000,A 180.000,B 0.000,C 180.000} C_DIS
LIN {X 108.053,Y 108.159,Z 67.000,A 180.000,B 0.000,C 180.000} C_DIS
LIN {X 108.159,Y 108.053,Z 67.000,A 180.000,B 0.000,C 180.000} C_DIS
LIN {X 108.565,Y 107.623,Z 67.000,A 180.000,B 0.000,C 180.000} C_DIS
LIN {X 108.695,Y 107.483,Z 67.000,A 180.000,B 0.000,C 180.000} C_DIS
LIN {X 108.729,Y 107.444,Z 67.000,A 180.000,B 0.000,C 180.000} C_DIS
LIN {X 109.182,Y 106.908,Z 67.000,A 180.000,B 0.000,C 180.000} C_DIS
LIN {X 109.232,Y 106.847,Z 67.000,A 180.000,B 0.000,C 180.000} C_DIS
LIN {X 109.322,Y 106.729,Z 67.000,A 180.000,B 0.000,C 180.000} C_DIS
LIN {X 109.591,Y 106.371,Z 67.000,A 180.000,B 0.000,C 180.000} C_DIS
LIN {X 109.724,Y 106.193,Z 67.000,A 180.000,B 0.000,C 180.000} C_DIS
LIN {X 109.768,Y 106.130,Z 67.000,A 180.000,B 0.000,C 180.000} C_DIS
LIN {X 109.846,Y 106.014,Z 67.000,A 180.000,B 0.000,C 180.000} C_DIS
LIN {X 110.126,Y 105.595,Z 67.000,A 180.000,B 0.000,C 180.000} C_DIS
LIN {X 110.203,Y 105.477,Z 67.000,A 180.000,B 0.000,C 180.000} C_DIS
LIN {X 110.304,Y 105.307,Z 67.000,A 180.000,B 0.000,C 180.000} C_DIS
LIN {X 110.520,Y 104.941,Z 67.000,A 180.000,B 0.000,C 180.000} C_DIS
LIN {X 110.625,Y 104.762,Z 67.000,A 180.000,B 0.000,C 180.000} C_DIS
LIN {X 110.662,Y 104.693,Z 67.000,A 180.000,B 0.000,C 180.000} C_DIS
LIN {X 110.903,Y 104.226,Z 67.000,A 180.000,B 0.000,C 180.000} C_DIS
LIN {X 110.995,Y 104.047,Z 67.000,A 180.000,B 0.000,C 180.000} C_DIS
LIN {X 111.019,Y 103.998,Z 67.000,A 180.000,B 0.000,C 180.000} C_DIS
LIN {X 111.078,Y 103.869,Z 67.000,A 180.000,B 0.000,C 180.000} C_DIS
LIN {X 111.318,Y 103.332,Z 67.000,A 180.000,B 0.000,C 180.000} C_DIS
LIN {X 111.377,Y 103.194,Z 67.000,A 180.000,B 0.000,C 180.000} C_DIS
LIN {X 111.392,Y 103.153,Z 67.000,A 180.000,B 0.000,C 180.000} C_DIS
LIN {X 111.597,Y 102.617,Z 67.000,A 180.000,B 0.000,C 180.000} C_DIS
LIN {X 111.664,Y 102.438,Z 67.000,A 180.000,B 0.000,C 180.000} C_DIS
LIN {X 111.721,Y 102.260,Z 67.000,A 180.000,B 0.000,C 180.000} C_DIS
LIN {X 111.892,Y 101.723,Z 67.000,A 180.000,B 0.000,C 180.000} C_DIS
LIN {X 111.913,Y 101.654,Z 67.000,A 180.000,B 0.000,C 180.000} C_DIS
LIN {X 111.943,Y 101.545,Z 67.000,A 180.000,B 0.000,C 180.000} C_DIS
LIN {X 112.092,Y 100.966,Z 67.000,A 180.000,B 0.000,C 180.000} C_DIS
LIN {X 112.126,Y 100.829,Z 67.000,A 180.000,B 0.000,C 180.000} C_DIS
LIN {X 112.162,Y 100.651,Z 67.000,A 180.000,B 0.000,C 180.000} C_DIS
LIN {X 112.271,Y 100.105,Z 67.000,A 180.000,B 0.000,C 180.000} C_DIS
LIN {X 112.300,Y 99.936,Z 67.000,A 180.000,B 0.000,C 180.000} C_DIS
LIN {X 112.376,Y 99.399,Z 67.000,A 180.000,B 0.000,C 180.000} C_DIS
LIN {X 112.401,Y 99.221,Z 67.000,A 180.000,B 0.000,C 180.000} C_DIS
LIN {X 112.418,Y 99.042,Z 67.000,A 180.000,B 0.000,C 180.000} C_DIS
LIN {X 112.464,Y 98.505,Z 67.000,A 180.000,B 0.000,C 180.000} C_DIS
LIN {X 112.477,Y 98.327,Z 67.000,A 180.000,B 0.000,C 180.000} C_DIS
LIN {X 112.483,Y 98.148,Z 67.000,A 180.000,B 0.000,C 180.000} C_DIS
LIN {X 112.498,Y 97.612,Z 67.000,A 180.000,B 0.000,C 180.000} C_DIS
LIN {X 112.499,Y 97.433,Z 67.000,A 180.000,B 0.000,C 180.000} C_DIS
LIN {X 112.484,Y 96.897,Z 67.000,A 180.000,B 0.000,C 180.000} C_DIS
LIN {X 112.479,Y 96.718,Z 67.000,A 180.000,B 0.000,C 180.000} C_DIS
LIN {X 112.467,Y 96.539,Z 67.000,A 180.000,B 0.000,C 180.000} C_DIS
LIN {X 112.422,Y 96.003,Z 67.000,A 180.000,B 0.000,C 180.000} C_DIS
LIN {X 112.406,Y 95.824,Z 67.000,A 180.000,B 0.000,C 180.000} C_DIS
LIN {X 112.382,Y 95.645,Z 67.000,A 180.000,B 0.000,C 180.000} C_DIS
LIN {X 112.306,Y 95.109,Z 67.000,A 180.000,B 0.000,C 180.000} C_DIS
LIN {X 112.278,Y 94.930,Z 67.000,A 180.000,B 0.000,C 180.000} C_DIS
LIN {X 112.271,Y 94.895,Z 67.000,A 180.000,B 0.000,C 180.000} C_DIS
LIN {X 112.171,Y 94.394,Z 67.000,A 180.000,B 0.000,C 180.000} C_DIS
LIN {X 112.135,Y 94.215,Z 67.000,A 180.000,B 0.000,C 180.000} C_DIS
LIN {X 112.092,Y 94.036,Z 67.000,A 180.000,B 0.000,C 180.000} C_DIS
LIN {X 111.954,Y 93.500,Z 67.000,A 180.000,B 0.000,C 180.000} C_DIS
LIN {X 111.913,Y 93.346,Z 67.000,A 180.000,B 0.000,C 180.000} C_DIS
LIN {X 111.906,Y 93.321,Z 67.000,A 180.000,B 0.000,C 180.000} C_DIS
LIN {X 111.849,Y 93.142,Z 67.000,A 180.000,B 0.000,C 180.000} C_DIS
LIN {X 111.734,Y 92.782,Z 67.000,A 180.000,B 0.000,C 180.000} C_DIS
LIN {X 111.678,Y 92.606,Z 67.000,A 180.000,B 0.000,C 180.000} C_DIS
LIN {X 111.614,Y 92.427,Z 67.000,A 180.000,B 0.000,C 180.000} C_DIS
LIN {X 111.409,Y 91.891,Z 67.000,A 180.000,B 0.000,C 180.000} C_DIS
LIN {X 111.377,Y 91.806,Z 67.000,A 180.000,B 0.000,C 180.000} C_DIS
LIN {X 111.338,Y 91.712,Z 67.000,A 180.000,B 0.000,C 180.000} C_DIS
LIN {X 111.258,Y 91.533,Z 67.000,A 180.000,B 0.000,C 180.000} C_DIS
LIN {X 111.098,Y 91.176,Z 67.000,A 180.000,B 0.000,C 180.000} C_DIS
LIN {X 111.019,Y 91.002,Z 67.000,A 180.000,B 0.000,C 180.000} C_DIS
LIN {X 111.017,Y 90.997,Z 67.000,A 180.000,B 0.000,C 180.000} C_DIS
LIN {X 110.926,Y 90.818,Z 67.000,A 180.000,B 0.000,C 180.000} C_DIS
LIN {X 110.662,Y 90.307,Z 67.000,A 180.000,B 0.000,C 180.000} C_DIS
LIN {X 110.649,Y 90.282,Z 67.000,A 180.000,B 0.000,C 180.000} C_DIS
LIN {X 110.546,Y 90.103,Z 67.000,A 180.000,B 0.000,C 180.000} C_DIS
LIN {X 110.304,Y 89.693,Z 67.000,A 180.000,B 0.000,C 180.000} C_DIS
LIN {X 110.230,Y 89.567,Z 67.000,A 180.000,B 0.000,C 180.000} C_DIS
LIN {X 110.126,Y 89.405,Z 67.000,A 180.000,B 0.000,C 180.000} C_DIS
LIN {X 109.875,Y 89.031,Z 67.000,A 180.000,B 0.000,C 180.000} C_DIS
LIN {X 109.768,Y 88.870,Z 67.000,A 180.000,B 0.000,C 180.000} C_DIS
LIN {X 109.756,Y 88.852,Z 67.000,A 180.000,B 0.000,C 180.000} C_DIS
LIN {X 109.624,Y 88.673,Z 67.000,A 180.000,B 0.000,C 180.000} C_DIS
LIN {X 109.355,Y 88.316,Z 67.000,A 180.000,B 0.000,C 180.000} C_DIS
LIN {X 109.232,Y 88.153,Z 67.000,A 180.000,B 0.000,C 180.000} C_DIS
LIN {X 109.219,Y 88.137,Z 67.000,A 180.000,B 0.000,C 180.000} C_DIS
LIN {X 109.069,Y 87.958,Z 67.000,A 180.000,B 0.000,C 180.000} C_DIS
LIN {X 108.767,Y 87.601,Z 67.000,A 180.000,B 0.000,C 180.000} C_DIS
LIN {X 108.695,Y 87.517,Z 67.000,A 180.000,B 0.000,C 180.000} C_DIS
LIN {X 108.607,Y 87.422,Z 67.000,A 180.000,B 0.000,C 180.000} C_DIS
LIN {X 108.159,Y 86.947,Z 67.000,A 180.000,B 0.000,C 180.000} C_DIS
LIN {X 108.099,Y 86.885,Z 67.000,A 180.000,B 0.000,C 180.000} C_DIS
LIN {X 107.980,Y 86.773,Z 67.000,A 180.000,B 0.000,C 180.000} C_DIS
LIN {X 107.623,Y 86.435,Z 67.000,A 180.000,B 0.000,C 180.000} C_DIS
LIN {X 107.532,Y 86.349,Z 67.000,A 180.000,B 0.000,C 180.000} C_DIS
LIN {X 107.444,Y 86.271,Z 67.000,A 180.000,B 0.000,C 180.000} C_DIS
LIN {X 106.908,Y 85.818,Z 67.000,A 180.000,B 0.000,C 180.000} C_DIS
LIN {X 106.902,Y 85.813,Z 67.000,A 180.000,B 0.000,C 180.000} C_DIS
LIN {X 106.729,Y 85.678,Z 67.000,A 180.000,B 0.000,C 180.000} C_DIS
LIN {X 106.371,Y 85.409,Z 67.000,A 180.000,B 0.000,C 180.000} C_DIS
LIN {X 106.194,Y 85.276,Z 67.000,A 180.000,B 0.000,C 180.000} C_DIS
LIN {X 106.193,Y 85.276,Z 67.000,A 180.000,B 0.000,C 180.000} C_DIS
LIN {X 106.014,Y 85.154,Z 67.000,A 180.000,B 0.000,C 180.000} C_DIS
LIN {X 105.656,Y 84.915,Z 67.000,A 180.000,B 0.000,C 180.000} C_DIS
LIN {X 105.477,Y 84.797,Z 67.000,A 180.000,B 0.000,C 180.000} C_DIS
LIN {X 105.382,Y 84.740,Z 67.000,A 180.000,B 0.000,C 180.000} C_DIS
LIN {X 104.941,Y 84.480,Z 67.000,A 180.000,B 0.000,C 180.000} C_DIS
LIN {X 104.775,Y 84.383,Z 67.000,A 180.000,B 0.000,C 180.000} C_DIS
LIN {X 104.762,Y 84.375,Z 67.000,A 180.000,B 0.000,C 180.000} C_DIS
LIN {X 104.584,Y 84.282,Z 67.000,A 180.000,B 0.000,C 180.000} C_DIS
LIN {X 104.087,Y 84.025,Z 67.000,A 180.000,B 0.000,C 180.000} C_DIS
LIN {X 104.047,Y 84.005,Z 67.000,A 180.000,B 0.000,C 180.000} C_DIS
LIN {X 103.869,Y 83.922,Z 67.000,A 180.000,B 0.000,C 180.000} C_DIS
LIN {X 103.300,Y 83.668,Z 67.000,A 180.000,B 0.000,C 180.000} C_DIS
LIN {X 103.153,Y 83.608,Z 67.000,A 180.000,B 0.000,C 180.000} C_DIS
LIN {X 102.617,Y 83.403,Z 67.000,A 180.000,B 0.000,C 180.000} C_DIS
LIN {X 102.438,Y 83.336,Z 67.000,A 180.000,B 0.000,C 180.000} C_DIS
LIN {X 102.358,Y 83.310,Z 67.000,A 180.000,B 0.000,C 180.000} C_DIS
LIN {X 101.723,Y 83.108,Z 67.000,A 180.000,B 0.000,C 180.000} C_DIS
LIN {X 101.545,Y 83.057,Z 67.000,A 180.000,B 0.000,C 180.000} C_DIS
LIN {X 101.008,Y 82.919,Z 67.000,A 180.000,B 0.000,C 180.000} C_DIS
LIN {X 100.829,Y 82.874,Z 67.000,A 180.000,B 0.000,C 180.000} C_DIS
LIN {X 100.651,Y 82.838,Z 67.000,A 180.000,B 0.000,C 180.000} C_DIS
LIN {X 100.114,Y 82.731,Z 67.000,A 180.000,B 0.000,C 180.000} C_DIS
LIN {X 99.936,Y 82.700,Z 67.000,A 180.000,B 0.000,C 180.000} C_DIS
LIN {X 99.399,Y 82.624,Z 67.000,A 180.000,B 0.000,C 180.000} C_DIS
LIN {X 99.221,Y 82.599,Z 67.000,A 180.000,B 0.000,C 180.000} C_DIS
LIN {X 99.185,Y 82.595,Z 67.000,A 180.000,B 0.000,C 180.000} C_DIS
LIN {X 99.042,Y 82.582,Z 67.000,A 180.000,B 0.000,C 180.000} C_DIS
LIN {X 98.505,Y 82.536,Z 67.000,A 180.000,B 0.000,C 180.000} C_DIS
LIN {X 98.327,Y 82.523,Z 67.000,A 180.000,B 0.000,C 180.000} C_DIS
LIN {X 98.148,Y 82.517,Z 67.000,A 180.000,B 0.000,C 180.000} C_DIS
LIN {X 97.612,Y 82.502,Z 67.000,A 180.000,B 0.000,C 180.000} C_DIS
LIN {X 97.433,Y 82.501,Z 67.000,A 180.000,B 0.000,C 180.000} C_DIS
LIN {X 96.897,Y 82.516,Z 67.000,A 180.000,B 0.000,C 180.000} C_DIS
LIN {X 96.718,Y 82.521,Z 67.000,A 180.000,B 0.000,C 180.000} C_DIS
LIN {X 96.539,Y 82.533,Z 67.000,A 180.000,B 0.000,C 180.000} C_DIS
LIN {X 96.003,Y 82.578,Z 67.000,A 180.000,B 0.000,C 180.000} C_DIS
LIN {X 95.824,Y 82.594,Z 67.000,A 180.000,B 0.000,C 180.000} C_DIS
LIN {X 95.815,Y 82.595,Z 67.000,A 180.000,B 0.000,C 180.000} C_DIS
LIN {X 95.645,Y 82.618,Z 67.000,A 180.000,B 0.000,C 180.000} C_DIS
LIN {X 95.109,Y 82.694,Z 67.000,A 180.000,B 0.000,C 180.000} C_DIS
LIN {X 94.930,Y 82.722,Z 67.000,A 180.000,B 0.000,C 180.000} C_DIS
LIN {X 94.751,Y 82.758,Z 67.000,A 180.000,B 0.000,C 180.000} C_DIS
LIN {X 94.394,Y 82.829,Z 67.000,A 180.000,B 0.000,C 180.000} C_DIS
LIN {X 94.215,Y 82.865,Z 67.000,A 180.000,B 0.000,C 180.000} C_DIS
LIN {X 94.036,Y 82.908,Z 67.000,A 180.000,B 0.000,C 180.000} C_DIS
LIN {X 93.500,Y 83.046,Z 67.000,A 180.000,B 0.000,C 180.000} C_DIS
LIN {X 93.321,Y 83.094,Z 67.000,A 180.000,B 0.000,C 180.000} C_DIS
LIN {X 93.203,Y 83.131,Z 67.000,A 180.000,B 0.000,C 180.000} C_DIS
LIN {X 92.642,Y 83.310,Z 67.000,A 180.000,B 0.000,C 180.000} C_DIS
LIN {X 92.606,Y 83.322,Z 67.000,A 180.000,B 0.000,C 180.000} C_DIS
LIN {X 92.427,Y 83.386,Z 67.000,A 180.000,B 0.000,C 180.000} C_DIS
LIN {X 91.891,Y 83.591,Z 67.000,A 180.000,B 0.000,C 180.000} C_DIS
LIN {X 91.712,Y 83.662,Z 67.000,A 180.000,B 0.000,C 180.000} C_DIS
LIN {X 91.700,Y 83.668,Z 67.000,A 180.000,B 0.000,C 180.000} C_DIS
LIN {X 91.176,Y 83.902,Z 67.000,A 180.000,B 0.000,C 180.000} C_DIS
LIN {X 90.997,Y 83.983,Z 67.000,A 180.000,B 0.000,C 180.000} C_DIS
LIN {X 90.913,Y 84.025,Z 67.000,A 180.000,B 0.000,C 180.000} C_DIS
LIN {X 90.461,Y 84.259,Z 67.000,A 180.000,B 0.000,C 180.000} C_DIS
LIN {X 90.282,Y 84.351,Z 67.000,A 180.000,B 0.000,C 180.000} C_DIS
LIN {X 90.225,Y 84.383,Z 67.000,A 180.000,B 0.000,C 180.000} C_DIS
LIN {X 90.103,Y 84.454,Z 67.000,A 180.000,B 0.000,C 180.000} C_DIS
LIN {X 89.618,Y 84.740,Z 67.000,A 180.000,B 0.000,C 180.000} C_DIS
LIN {X 89.567,Y 84.770,Z 67.000,A 180.000,B 0.000,C 180.000} C_DIS
LIN {X 89.388,Y 84.886,Z 67.000,A 180.000,B 0.000,C 180.000} C_DIS
LIN {X 89.031,Y 85.125,Z 67.000,A 180.000,B 0.000,C 180.000} C_DIS
LIN {X 88.852,Y 85.244,Z 67.000,A 180.000,B 0.000,C 180.000} C_DIS
LIN {X 88.806,Y 85.276,Z 67.000,A 180.000,B 0.000,C 180.000} C_DIS
LIN {X 88.673,Y 85.376,Z 67.000,A 180.000,B 0.000,C 180.000} C_DIS
LIN {X 88.316,Y 85.645,Z 67.000,A 180.000,B 0.000,C 180.000} C_DIS
LIN {X 88.137,Y 85.781,Z 67.000,A 180.000,B 0.000,C 180.000} C_DIS
LIN {X 88.098,Y 85.813,Z 67.000,A 180.000,B 0.000,C 180.000} C_DIS
LIN {X 87.779,Y 86.082,Z 67.000,A 180.000,B 0.000,C 180.000} C_DIS
LIN {X 87.601,Y 86.233,Z 67.000,A 180.000,B 0.000,C 180.000} C_DIS
LIN {X 87.468,Y 86.349,Z 67.000,A 180.000,B 0.000,C 180.000} C_DIS
LIN {X 87.422,Y 86.393,Z 67.000,A 180.000,B 0.000,C 180.000} C_DIS
LIN {X 87.064,Y 86.731,Z 67.000,A 180.000,B 0.000,C 180.000} C_DIS
LIN {X 86.901,Y 86.885,Z 67.000,A 180.000,B 0.000,C 180.000} C_DIS
LIN {X 86.885,Y 86.901,Z 67.000,A 180.000,B 0.000,C 180.000} C_DIS
LIN {X 86.731,Y 87.064,Z 67.000,A 180.000,B 0.000,C 180.000} C_DIS
LIN {X 86.393,Y 87.422,Z 67.000,A 180.000,B 0.000,C 180.000} C_DIS
LIN {X 86.349,Y 87.468,Z 67.000,A 180.000,B 0.000,C 180.000} C_DIS
LIN {X 86.233,Y 87.601,Z 67.000,A 180.000,B 0.000,C 180.000} C_DIS
LIN {X 85.931,Y 87.958,Z 67.000,A 180.000,B 0.000,C 180.000} C_DIS
LIN {X 85.813,Y 88.098,Z 67.000,A 180.000,B 0.000,C 180.000} C_DIS
LIN {X 85.781,Y 88.137,Z 67.000,A 180.000,B 0.000,C 180.000} C_DIS
LIN {X 85.645,Y 88.316,Z 67.000,A 180.000,B 0.000,C 180.000} C_DIS
LIN {X 85.376,Y 88.673,Z 67.000,A 180.000,B 0.000,C 180.000} C_DIS
LIN {X 85.276,Y 88.806,Z 67.000,A 180.000,B 0.000,C 180.000} C_DIS
LIN {X 85.244,Y 88.852,Z 67.000,A 180.000,B 0.000,C 180.000} C_DIS
LIN {X 85.125,Y 89.031,Z 67.000,A 180.000,B 0.000,C 180.000} C_DIS
LIN {X 84.886,Y 89.388,Z 67.000,A 180.000,B 0.000,C 180.000} C_DIS
LIN {X 84.770,Y 89.567,Z 67.000,A 180.000,B 0.000,C 180.000} C_DIS
LIN {X 84.740,Y 89.618,Z 67.000,A 180.000,B 0.000,C 180.000} C_DIS
LIN {X 84.454,Y 90.103,Z 67.000,A 180.000,B 0.000,C 180.000} C_DIS
LIN {X 84.383,Y 90.225,Z 67.000,A 180.000,B 0.000,C 180.000} C_DIS
LIN {X 84.351,Y 90.282,Z 67.000,A 180.000,B 0.000,C 180.000} C_DIS
LIN {X 84.259,Y 90.461,Z 67.000,A 180.000,B 0.000,C 180.000} C_DIS
LIN {X 84.025,Y 90.913,Z 67.000,A 180.000,B 0.000,C 180.000} C_DIS
LIN {X 83.983,Y 90.997,Z 67.000,A 180.000,B 0.000,C 180.000} C_DIS
LIN {X 83.902,Y 91.176,Z 67.000,A 180.000,B 0.000,C 180.000} C_DIS
LIN {X 83.668,Y 91.700,Z 67.000,A 180.000,B 0.000,C 180.000} C_DIS
LIN {X 83.662,Y 91.712,Z 67.000,A 180.000,B 0.000,C 180.000} C_DIS
LIN {X 83.591,Y 91.891,Z 67.000,A 180.000,B 0.000,C 180.000} C_DIS
LIN {X 83.386,Y 92.427,Z 67.000,A 180.000,B 0.000,C 180.000} C_DIS
LIN {X 83.322,Y 92.606,Z 67.000,A 180.000,B 0.000,C 180.000} C_DIS
LIN {X 83.310,Y 92.642,Z 67.000,A 180.000,B 0.000,C 180.000} C_DIS
LIN {X 83.131,Y 93.203,Z 67.000,A 180.000,B 0.000,C 180.000} C_DIS
LIN {X 83.094,Y 93.321,Z 67.000,A 180.000,B 0.000,C 180.000} C_DIS
LIN {X 83.046,Y 93.500,Z 67.000,A 180.000,B 0.000,C 180.000} C_DIS
LIN {X 82.908,Y 94.036,Z 67.000,A 180.000,B 0.000,C 180.000} C_DIS
LIN {X 82.865,Y 94.215,Z 67.000,A 180.000,B 0.000,C 180.000} C_DIS
LIN {X 82.829,Y 94.394,Z 67.000,A 180.000,B 0.000,C 180.000} C_DIS
LIN {X 82.758,Y 94.751,Z 67.000,A 180.000,B 0.000,C 180.000} C_DIS
LIN {X 82.722,Y 94.930,Z 67.000,A 180.000,B 0.000,C 180.000} C_DIS
LIN {X 82.694,Y 95.109,Z 67.000,A 180.000,B 0.000,C 180.000} C_DIS
LIN {X 82.618,Y 95.645,Z 67.000,A 180.000,B 0.000,C 180.000} C_DIS
LIN {X 82.595,Y 95.815,Z 67.000,A 180.000,B 0.000,C 180.000} C_DIS
LIN {X 82.594,Y 95.824,Z 67.000,A 180.000,B 0.000,C 180.000} C_DIS
LIN {X 82.589,Y 95.875,Z 67.000,A 180.000,B 0.000,C 180.000} C_DIS
; Link Move Starts
LIN {X 82.562,Y 96.189,Z 67.000,A 180.000,B 0.000,C 180.000} C_DIS
LIN {X 82.536,Y 96.503,Z 66.998,A 180.000,B 0.000,C 180.000} C_DIS
LIN {X 82.518,Y 96.817,Z 66.996,A 180.000,B 0.000,C 180.000} C_DIS
LIN {X 82.509,Y 97.132,Z 66.992,A 180.000,B 0.000,C 180.000} C_DIS
LIN {X 82.501,Y 97.447,Z 66.988,A 180.000,B 0.000,C 180.000} C_DIS
LIN {X 82.506,Y 97.762,Z 66.983,A 180.000,B 0.000,C 180.000} C_DIS
LIN {X 82.511,Y 97.919,Z 66.981,A 180.000,B 0.000,C 180.000} C_DIS
LIN {X 82.515,Y 98.077,Z 66.978,A 180.000,B 0.000,C 180.000} C_DIS
LIN {X 82.520,Y 98.234,Z 66.975,A 180.000,B 0.000,C 180.000} C_DIS
LIN {X 82.527,Y 98.392,Z 66.971,A 180.000,B 0.000,C 180.000} C_DIS
LIN {X 82.540,Y 98.549,Z 66.968,A 180.000,B 0.000,C 180.000} C_DIS
LIN {X 82.553,Y 98.706,Z 66.964,A 180.000,B 0.000,C 180.000} C_DIS
LIN {X 82.567,Y 98.862,Z 66.960,A 180.000,B 0.000,C 180.000} C_DIS
LIN {X 82.580,Y 99.019,Z 66.956,A 180.000,B 0.000,C 180.000} C_DIS
LIN {X 82.594,Y 99.176,Z 66.952,A 180.000,B 0.000,C 180.000} C_DIS
LIN {X 82.615,Y 99.332,Z 66.948,A 180.000,B 0.000,C 180.000} C_DIS
LIN {X 82.637,Y 99.488,Z 66.944,A 180.000,B 0.000,C 180.000} C_DIS
LIN {X 82.659,Y 99.644,Z 66.939,A 180.000,B 0.000,C 180.000} C_DIS
LIN {X 82.681,Y 99.800,Z 66.934,A 180.000,B 0.000,C 180.000} C_DIS
LIN {X 82.703,Y 99.956,Z 66.929,A 180.000,B 0.000,C 180.000} C_DIS
LIN {X 82.731,Y 100.111,Z 66.924,A 180.000,B 0.000,C 180.000} C_DIS
LIN {X 82.746,Y 100.188,Z 66.922,A 180.000,B 0.000,C 180.000} C_DIS
LIN {X 82.761,Y 100.266,Z 66.919,A 180.000,B 0.000,C 180.000} C_DIS
LIN {X 82.777,Y 100.343,Z 66.917,A 180.000,B 0.000,C 180.000} C_DIS
LIN {X 82.792,Y 100.420,Z 66.914,A 180.000,B 0.000,C 180.000} C_DIS
LIN {X 82.807,Y 100.497,Z 66.911,A 180.000,B 0.000,C 180.000} C_DIS
LIN {X 82.823,Y 100.575,Z 66.909,A 180.000,B 0.000,C 180.000} C_DIS
LIN {X 82.838,Y 100.652,Z 66.906,A 180.000,B 0.000,C 180.000} C_DIS
LIN {X 82.853,Y 100.729,Z 66.903,A 180.000,B 0.000,C 180.000} C_DIS
LIN {X 82.869,Y 100.806,Z 66.901,A 180.000,B 0.000,C 180.000} C_DIS
LIN {X 82.887,Y 100.883,Z 66.898,A 180.000,B 0.000,C 180.000} C_DIS
LIN {X 82.906,Y 100.959,Z 66.895,A 180.000,B 0.000,C 180.000} C_DIS
LIN {X 82.926,Y 101.036,Z 66.892,A 180.000,B 0.000,C 180.000} C_DIS
LIN {X 82.946,Y 101.112,Z 66.890,A 180.000,B 0.000,C 180.000} C_DIS
LIN {X 82.965,Y 101.188,Z 66.887,A 180.000,B 0.000,C 180.000} C_DIS
LIN {X 82.985,Y 101.264,Z 66.884,A 180.000,B 0.000,C 180.000} C_DIS
LIN {X 83.005,Y 101.341,Z 66.881,A 180.000,B 0.000,C 180.000} C_DIS
LIN {X 83.024,Y 101.417,Z 66.878,A 180.000,B 0.000,C 180.000} C_DIS
LIN {X 83.044,Y 101.493,Z 66.876,A 180.000,B 0.000,C 180.000} C_DIS
LIN {X 83.064,Y 101.569,Z 66.873,A 180.000,B 0.000,C 180.000} C_DIS
LIN {X 83.084,Y 101.645,Z 66.870,A 180.000,B 0.000,C 180.000} C_DIS
LIN {X 83.107,Y 101.721,Z 66.867,A 180.000,B 0.000,C 180.000} C_DIS
LIN {X 83.131,Y 101.796,Z 66.865,A 180.000,B 0.000,C 180.000} C_DIS
LIN {X 83.155,Y 101.871,Z 66.862,A 180.000,B 0.000,C 180.000} C_DIS
LIN {X 83.203,Y 102.021,Z 66.856,A 180.000,B 0.000,C 180.000} C_DIS
LIN {X 83.227,Y 102.096,Z 66.854,A 180.000,B 0.000,C 180.000} C_DIS
LIN {X 83.274,Y 102.246,Z 66.848,A 180.000,B 0.000,C 180.000} C_DIS
LIN {X 83.298,Y 102.321,Z 66.845,A 180.000,B 0.000,C 180.000} C_DIS
LIN {X 83.322,Y 102.396,Z 66.843,A 180.000,B 0.000,C 180.000} C_DIS
LIN {X 83.348,Y 102.471,Z 66.840,A 180.000,B 0.000,C 180.000} C_DIS
LIN {X 83.375,Y 102.544,Z 66.837,A 180.000,B 0.000,C 180.000} C_DIS
LIN {X 83.459,Y 102.765,Z 66.829,A 180.000,B 0.000,C 180.000} C_DIS
LIN {X 83.516,Y 102.912,Z 66.823,A 180.000,B 0.000,C 180.000} C_DIS
LIN {X 83.544,Y 102.986,Z 66.821,A 180.000,B 0.000,C 180.000} C_DIS
LIN {X 83.600,Y 103.133,Z 66.815,A 180.000,B 0.000,C 180.000} C_DIS
LIN {X 83.628,Y 103.207,Z 66.812,A 180.000,B 0.000,C 180.000} C_DIS
LIN {X 83.658,Y 103.279,Z 66.810,A 180.000,B 0.000,C 180.000} C_DIS
LIN {X 83.690,Y 103.351,Z 66.807,A 180.000,B 0.000,C 180.000} C_DIS
LIN {X 83.755,Y 103.495,Z 66.801,A 180.000,B 0.000,C 180.000} C_DIS
LIN {X 83.787,Y 103.567,Z 66.799,A 180.000,B 0.000,C 180.000} C_DIS
LIN {X 83.851,Y 103.711,Z 66.793,A 180.000,B 0.000,C 180.000} C_DIS
LIN {X 83.948,Y 103.926,Z 66.785,A 180.000,B 0.000,C 180.000} C_DIS
LIN {X 83.980,Y 103.998,Z 66.782,A 180.000,B 0.000,C 180.000} C_DIS
LIN {X 84.015,Y 104.068,Z 66.779,A 180.000,B 0.000,C 180.000} C_DIS
LIN {X 84.124,Y 104.278,Z 66.771,A 180.000,B 0.000,C 180.000} C_DIS
LIN {X 84.341,Y 104.698,Z 66.755,A 180.000,B 0.000,C 180.000} C_DIS
LIN {X 84.378,Y 104.767,Z 66.752,A 180.000,B 0.000,C 180.000} C_DIS
LIN {X 84.418,Y 104.836,Z 66.749,A 180.000,B 0.000,C 180.000} C_DIS
LIN {X 84.738,Y 105.378,Z 66.727,A 180.000,B 0.000,C 180.000} C_DIS
LIN {X 84.778,Y 105.446,Z 66.724,A 180.000,B 0.000,C 180.000} C_DIS
LIN {X 84.820,Y 105.513,Z 66.722,A 180.000,B 0.000,C 180.000} C_DIS
LIN {X 84.863,Y 105.578,Z 66.719,A 180.000,B 0.000,C 180.000} C_DIS
LIN {X 85.126,Y 105.971,Z 66.702,A 180.000,B 0.000,C 180.000} C_DIS
LIN {X 85.170,Y 106.037,Z 66.700,A 180.000,B 0.000,C 180.000} C_DIS
LIN {X 85.213,Y 106.102,Z 66.697,A 180.000,B 0.000,C 180.000} C_DIS
LIN {X 85.258,Y 106.167,Z 66.694,A 180.000,B 0.000,C 180.000} C_DIS
LIN {X 85.304,Y 106.231,Z 66.691,A 180.000,B 0.000,C 180.000} C_DIS
LIN {X 85.351,Y 106.294,Z 66.689,A 180.000,B 0.000,C 180.000} C_DIS
LIN {X 85.446,Y 106.420,Z 66.683,A 180.000,B 0.000,C 180.000} C_DIS
LIN {X 85.588,Y 106.609,Z 66.675,A 180.000,B 0.000,C 180.000} C_DIS
LIN {X 85.683,Y 106.734,Z 66.669,A 180.000,B 0.000,C 180.000} C_DIS
LIN {X 85.730,Y 106.797,Z 66.667,A 180.000,B 0.000,C 180.000} C_DIS
LIN {X 85.778,Y 106.859,Z 66.664,A 180.000,B 0.000,C 180.000} C_DIS
LIN {X 85.828,Y 106.920,Z 66.661,A 180.000,B 0.000,C 180.000} C_DIS
LIN {X 85.981,Y 107.101,Z 66.653,A 180.000,B 0.000,C 180.000} C_DIS
LIN {X 86.083,Y 107.221,Z 66.647,A 180.000,B 0.000,C 180.000} C_DIS
LIN {X 86.133,Y 107.281,Z 66.645,A 180.000,B 0.000,C 180.000} C_DIS
LIN {X 86.235,Y 107.401,Z 66.639,A 180.000,B 0.000,C 180.000} C_DIS
LIN {X 86.286,Y 107.462,Z 66.636,A 180.000,B 0.000,C 180.000} C_DIS
LIN {X 86.338,Y 107.520,Z 66.634,A 180.000,B 0.000,C 180.000} C_DIS
LIN {X 86.392,Y 107.578,Z 66.631,A 180.000,B 0.000,C 180.000} C_DIS
LIN {X 86.446,Y 107.635,Z 66.628,A 180.000,B 0.000,C 180.000} C_DIS
LIN {X 86.500,Y 107.692,Z 66.625,A 180.000,B 0.000,C 180.000} C_DIS
LIN {X 86.554,Y 107.749,Z 66.623,A 180.000,B 0.000,C 180.000} C_DIS
LIN {X 86.609,Y 107.807,Z 66.620,A 180.000,B 0.000,C 180.000} C_DIS
LIN {X 86.663,Y 107.864,Z 66.617,A 180.000,B 0.000,C 180.000} C_DIS
LIN {X 86.717,Y 107.921,Z 66.614,A 180.000,B 0.000,C 180.000} C_DIS
LIN {X 86.771,Y 107.978,Z 66.612,A 180.000,B 0.000,C 180.000} C_DIS
LIN {X 86.825,Y 108.036,Z 66.609,A 180.000,B 0.000,C 180.000} C_DIS
LIN {X 86.879,Y 108.092,Z 66.606,A 180.000,B 0.000,C 180.000} C_DIS
LIN {X 86.936,Y 108.148,Z 66.603,A 180.000,B 0.000,C 180.000} C_DIS
LIN {X 86.993,Y 108.202,Z 66.601,A 180.000,B 0.000,C 180.000} C_DIS
LIN {X 87.050,Y 108.256,Z 66.598,A 180.000,B 0.000,C 180.000} C_DIS
LIN {X 87.107,Y 108.310,Z 66.595,A 180.000,B 0.000,C 180.000} C_DIS
LIN {X 87.164,Y 108.364,Z 66.592,A 180.000,B 0.000,C 180.000} C_DIS
LIN {X 87.222,Y 108.418,Z 66.590,A 180.000,B 0.000,C 180.000} C_DIS
LIN {X 87.279,Y 108.472,Z 66.587,A 180.000,B 0.000,C 180.000} C_DIS
LIN {X 87.336,Y 108.526,Z 66.584,A 180.000,B 0.000,C 180.000} C_DIS
LIN {X 87.393,Y 108.581,Z 66.582,A 180.000,B 0.000,C 180.000} C_DIS
LIN {X 87.451,Y 108.635,Z 66.579,A 180.000,B 0.000,C 180.000} C_DIS
LIN {X 87.509,Y 108.688,Z 66.577,A 180.000,B 0.000,C 180.000} C_DIS
LIN {X 87.568,Y 108.739,Z 66.574,A 180.000,B 0.000,C 180.000} C_DIS
LIN {X 87.688,Y 108.841,Z 66.569,A 180.000,B 0.000,C 180.000} C_DIS
LIN {X 87.809,Y 108.943,Z 66.564,A 180.000,B 0.000,C 180.000} C_DIS
LIN {X 87.929,Y 109.044,Z 66.560,A 180.000,B 0.000,C 180.000} C_DIS
LIN {X 88.049,Y 109.146,Z 66.555,A 180.000,B 0.000,C 180.000} C_DIS
LIN {X 88.171,Y 109.246,Z 66.551,A 180.000,B 0.000,C 180.000} C_DIS
LIN {X 88.297,Y 109.341,Z 66.547,A 180.000,B 0.000,C 180.000} C_DIS
LIN {X 88.423,Y 109.436,Z 66.542,A 180.000,B 0.000,C 180.000} C_DIS
LIN {X 88.548,Y 109.530,Z 66.539,A 180.000,B 0.000,C 180.000} C_DIS
LIN {X 88.674,Y 109.625,Z 66.535,A 180.000,B 0.000,C 180.000} C_DIS
LIN {X 88.800,Y 109.719,Z 66.531,A 180.000,B 0.000,C 180.000} C_DIS
LIN {X 88.930,Y 109.808,Z 66.528,A 180.000,B 0.000,C 180.000} C_DIS
LIN {X 89.061,Y 109.896,Z 66.524,A 180.000,B 0.000,C 180.000} C_DIS
LIN {X 89.192,Y 109.983,Z 66.521,A 180.000,B 0.000,C 180.000} C_DIS
LIN {X 89.323,Y 110.071,Z 66.519,A 180.000,B 0.000,C 180.000} C_DIS
LIN {X 89.454,Y 110.158,Z 66.516,A 180.000,B 0.000,C 180.000} C_DIS
LIN {X 89.723,Y 110.322,Z 66.511,A 180.000,B 0.000,C 180.000} C_DIS
LIN {X 89.994,Y 110.482,Z 66.507,A 180.000,B 0.000,C 180.000} C_DIS
LIN {X 90.267,Y 110.641,Z 66.504,A 180.000,B 0.000,C 180.000} C_DIS
LIN {X 90.546,Y 110.786,Z 66.502,A 180.000,B 0.000,C 180.000} C_DIS
LIN {X 90.826,Y 110.930,Z 66.500,A 180.000,B 0.000,C 180.000} C_DIS
LIN {X 91.070,Y 111.050,Z 66.500,A 180.000,B 0.000,C 180.000} C_DIS
; Cutting Move Starts
LIN {X 91.176,Y 111.098,Z 66.500,A 180.000,B 0.000,C 180.000} C_DIS
LIN {X 91.533,Y 111.258,Z 66.500,A 180.000,B 0.000,C 180.000} C_DIS
LIN {X 91.712,Y 111.338,Z 66.500,A 180.000,B 0.000,C 180.000} C_DIS
LIN {X 91.806,Y 111.377,Z 66.500,A 180.000,B 0.000,C 180.000} C_DIS
LIN {X 91.891,Y 111.409,Z 66.500,A 180.000,B 0.000,C 180.000} C_DIS
LIN {X 92.427,Y 111.614,Z 66.500,A 180.000,B 0.000,C 180.000} C_DIS
LIN {X 92.606,Y 111.678,Z 66.500,A 180.000,B 0.000,C 180.000} C_DIS
LIN {X 92.964,Y 111.792,Z 66.500,A 180.000,B 0.000,C 180.000} C_DIS
LIN {X 93.142,Y 111.849,Z 66.500,A 180.000,B 0.000,C 180.000} C_DIS
LIN {X 93.321,Y 111.906,Z 66.500,A 180.000,B 0.000,C 180.000} C_DIS
LIN {X 93.346,Y 111.913,Z 66.500,A 180.000,B 0.000,C 180.000} C_DIS
LIN {X 93.500,Y 111.954,Z 66.500,A 180.000,B 0.000,C 180.000} C_DIS
LIN {X 94.036,Y 112.092,Z 66.500,A 180.000,B 0.000,C 180.000} C_DIS
LIN {X 94.215,Y 112.135,Z 66.500,A 180.000,B 0.000,C 180.000} C_DIS
LIN {X 94.394,Y 112.171,Z 66.500,A 180.000,B 0.000,C 180.000} C_DIS
LIN {X 94.895,Y 112.271,Z 66.500,A 180.000,B 0.000,C 180.000} C_DIS
LIN {X 94.930,Y 112.278,Z 66.500,A 180.000,B 0.000,C 180.000} C_DIS
LIN {X 95.109,Y 112.306,Z 66.500,A 180.000,B 0.000,C 180.000} C_DIS
LIN {X 95.645,Y 112.382,Z 66.500,A 180.000,B 0.000,C 180.000} C_DIS
LIN {X 95.824,Y 112.406,Z 66.500,A 180.000,B 0.000,C 180.000} C_DIS
LIN {X 96.003,Y 112.422,Z 66.500,A 180.000,B 0.000,C 180.000} C_DIS
LIN {X 96.539,Y 112.467,Z 66.500,A 180.000,B 0.000,C 180.000} C_DIS
LIN {X 96.718,Y 112.479,Z 66.500,A 180.000,B 0.000,C 180.000} C_DIS
LIN {X 96.897,Y 112.484,Z 66.500,A 180.000,B 0.000,C 180.000} C_DIS
LIN {X 97.433,Y 112.499,Z 66.500,A 180.000,B 0.000,C 180.000} C_DIS
LIN {X 97.612,Y 112.498,Z 66.500,A 180.000,B 0.000,C 180.000} C_DIS
LIN {X 98.148,Y 112.483,Z 66.500,A 180.000,B 0.000,C 180.000} C_DIS
LIN {X 98.327,Y 112.477,Z 66.500,A 180.000,B 0.000,C 180.000} C_DIS
LIN {X 98.505,Y 112.464,Z 66.500,A 180.000,B 0.000,C 180.000} C_DIS
LIN {X 99.042,Y 112.418,Z 66.500,A 180.000,B 0.000,C 180.000} C_DIS
LIN {X 99.221,Y 112.401,Z 66.500,A 180.000,B 0.000,C 180.000} C_DIS
LIN {X 99.399,Y 112.376,Z 66.500,A 180.000,B 0.000,C 180.000} C_DIS
LIN {X 99.936,Y 112.300,Z 66.500,A 180.000,B 0.000,C 180.000} C_DIS
LIN {X 100.105,Y 112.271,Z 66.500,A 180.000,B 0.000,C 180.000} C_DIS
LIN {X 100.651,Y 112.162,Z 66.500,A 180.000,B 0.000,C 180.000} C_DIS
LIN {X 100.829,Y 112.126,Z 66.500,A 180.000,B 0.000,C 180.000} C_DIS
LIN {X 100.966,Y 112.092,Z 66.500,A 180.000,B 0.000,C 180.000} C_DIS
LIN {X 101.545,Y 111.943,Z 66.500,A 180.000,B 0.000,C 180.000} C_DIS
LIN {X 101.654,Y 111.913,Z 66.500,A 180.000,B 0.000,C 180.000} C_DIS
LIN {X 101.723,Y 111.892,Z 66.500,A 180.000,B 0.000,C 180.000} C_DIS
LIN {X 102.260,Y 111.721,Z 66.500,A 180.000,B 0.000,C 180.000} C_DIS
LIN {X 102.438,Y 111.664,Z 66.500,A 180.000,B 0.000,C 180.000} C_DIS
LIN {X 102.617,Y 111.597,Z 66.500,A 180.000,B 0.000,C 180.000} C_DIS
LIN {X 103.153,Y 111.392,Z 66.500,A 180.000,B 0.000,C 180.000} C_DIS
LIN {X 103.194,Y 111.377,Z 66.500,A 180.000,B 0.000,C 180.000} C_DIS
LIN {X 103.332,Y 111.318,Z 66.500,A 180.000,B 0.000,C 180.000} C_DIS
LIN {X 103.869,Y 111.078,Z 66.500,A 180.000,B 0.000,C 180.000} C_DIS
LIN {X 103.998,Y 111.019,Z 66.500,A 180.000,B 0.000,C 180.000} C_DIS
LIN {X 104.047,Y 110.995,Z 66.500,A 180.000,B 0.000,C 180.000} C_DIS
LIN {X 104.226,Y 110.903,Z 66.500,A 180.000,B 0.000,C 180.000} C_DIS
LIN {X 104.693,Y 110.662,Z 66.500,A 180.000,B 0.000,C 180.000} C_DIS
LIN {X 104.762,Y 110.625,Z 66.500,A 180.000,B 0.000,C 180.000} C_DIS
LIN {X 104.941,Y 110.520,Z 66.500,A 180.000,B 0.000,C 180.000} C_DIS
LIN {X 105.307,Y 110.304,Z 66.500,A 180.000,B 0.000,C 180.000} C_DIS
LIN {X 105.477,Y 110.203,Z 66.500,A 180.000,B 0.000,C 180.000} C_DIS
LIN {X 105.595,Y 110.126,Z 66.500,A 180.000,B 0.000,C 180.000} C_DIS
LIN {X 106.014,Y 109.846,Z 66.500,A 180.000,B 0.000,C 180.000} C_DIS
LIN {X 106.130,Y 109.768,Z 66.500,A 180.000,B 0.000,C 180.000} C_DIS
LIN {X 106.193,Y 109.724,Z 66.500,A 180.000,B 0.000,C 180.000} C_DIS
LIN {X 106.371,Y 109.591,Z 66.500,A 180.000,B 0.000,C 180.000} C_DIS
LIN {X 106.729,Y 109.322,Z 66.500,A 180.000,B 0.000,C 180.000} C_DIS
LIN {X 106.847,Y 109.232,Z 66.500,A 180.000,B 0.000,C 180.000} C_DIS
LIN {X 106.908,Y 109.182,Z 66.500,A 180.000,B 0.000,C 180.000} C_DIS
LIN {X 107.444,Y 108.729,Z 66.500,A 180.000,B 0.000,C 180.000} C_DIS
LIN {X 107.483,Y 108.695,Z 66.500,A 180.000,B 0.000,C 180.000} C_DIS
LIN {X 107.623,Y 108.565,Z 66.500,A 180.000,B 0.000,C 180.000} C_DIS
LIN {X 108.053,Y 108.159,Z 66.500,A 180.000,B 0.000,C 180.000} C_DIS
LIN {X 108.159,Y 108.053,Z 66.500,A 180.000,B 0.000,C 180.000} C_DIS
LIN {X 108.565,Y 107.623,Z 66.500,A 180.000,B 0.000,C 180.000} C_DIS
LIN {X 108.695,Y 107.483,Z 66.500,A 180.000,B 0.000,C 180.000} C_DIS
LIN {X 108.729,Y 107.444,Z 66.500,A 180.000,B 0.000,C 180.000} C_DIS
LIN {X 109.182,Y 106.908,Z 66.500,A 180.000,B 0.000,C 180.000} C_DIS
LIN {X 109.232,Y 106.847,Z 66.500,A 180.000,B 0.000,C 180.000} C_DIS
LIN {X 109.322,Y 106.729,Z 66.500,A 180.000,B 0.000,C 180.000} C_DIS
LIN {X 109.591,Y 106.371,Z 66.500,A 180.000,B 0.000,C 180.000} C_DIS
LIN {X 109.724,Y 106.193,Z 66.500,A 180.000,B 0.000,C 180.000} C_DIS
LIN {X 109.768,Y 106.130,Z 66.500,A 180.000,B 0.000,C 180.000} C_DIS
LIN {X 109.846,Y 106.014,Z 66.500,A 180.000,B 0.000,C 180.000} C_DIS
LIN {X 110.126,Y 105.595,Z 66.500,A 180.000,B 0.000,C 180.000} C_DIS
LIN {X 110.203,Y 105.477,Z 66.500,A 180.000,B 0.000,C 180.000} C_DIS
LIN {X 110.304,Y 105.307,Z 66.500,A 180.000,B 0.000,C 180.000} C_DIS
LIN {X 110.520,Y 104.941,Z 66.500,A 180.000,B 0.000,C 180.000} C_DIS
LIN {X 110.625,Y 104.762,Z 66.500,A 180.000,B 0.000,C 180.000} C_DIS
LIN {X 110.662,Y 104.693,Z 66.500,A 180.000,B 0.000,C 180.000} C_DIS
LIN {X 110.903,Y 104.226,Z 66.500,A 180.000,B 0.000,C 180.000} C_DIS
LIN {X 110.995,Y 104.047,Z 66.500,A 180.000,B 0.000,C 180.000} C_DIS
LIN {X 111.019,Y 103.998,Z 66.500,A 180.000,B 0.000,C 180.000} C_DIS
LIN {X 111.078,Y 103.869,Z 66.500,A 180.000,B 0.000,C 180.000} C_DIS
LIN {X 111.318,Y 103.332,Z 66.500,A 180.000,B 0.000,C 180.000} C_DIS
LIN {X 111.377,Y 103.194,Z 66.500,A 180.000,B 0.000,C 180.000} C_DIS
LIN {X 111.392,Y 103.153,Z 66.500,A 180.000,B 0.000,C 180.000} C_DIS
LIN {X 111.597,Y 102.617,Z 66.500,A 180.000,B 0.000,C 180.000} C_DIS
LIN {X 111.664,Y 102.438,Z 66.500,A 180.000,B 0.000,C 180.000} C_DIS
LIN {X 111.721,Y 102.260,Z 66.500,A 180.000,B 0.000,C 180.000} C_DIS
LIN {X 111.892,Y 101.723,Z 66.500,A 180.000,B 0.000,C 180.000} C_DIS
LIN {X 111.913,Y 101.654,Z 66.500,A 180.000,B 0.000,C 180.000} C_DIS
LIN {X 111.943,Y 101.545,Z 66.500,A 180.000,B 0.000,C 180.000} C_DIS
LIN {X 112.092,Y 100.966,Z 66.500,A 180.000,B 0.000,C 180.000} C_DIS
LIN {X 112.126,Y 100.829,Z 66.500,A 180.000,B 0.000,C 180.000} C_DIS
LIN {X 112.162,Y 100.651,Z 66.500,A 180.000,B 0.000,C 180.000} C_DIS
LIN {X 112.271,Y 100.105,Z 66.500,A 180.000,B 0.000,C 180.000} C_DIS
LIN {X 112.300,Y 99.936,Z 66.500,A 180.000,B 0.000,C 180.000} C_DIS
LIN {X 112.376,Y 99.399,Z 66.500,A 180.000,B 0.000,C 180.000} C_DIS
LIN {X 112.401,Y 99.221,Z 66.500,A 180.000,B 0.000,C 180.000} C_DIS
LIN {X 112.418,Y 99.042,Z 66.500,A 180.000,B 0.000,C 180.000} C_DIS
LIN {X 112.464,Y 98.505,Z 66.500,A 180.000,B 0.000,C 180.000} C_DIS
LIN {X 112.477,Y 98.327,Z 66.500,A 180.000,B 0.000,C 180.000} C_DIS
LIN {X 112.483,Y 98.148,Z 66.500,A 180.000,B 0.000,C 180.000} C_DIS
LIN {X 112.498,Y 97.612,Z 66.500,A 180.000,B 0.000,C 180.000} C_DIS
LIN {X 112.499,Y 97.433,Z 66.500,A 180.000,B 0.000,C 180.000} C_DIS
LIN {X 112.484,Y 96.897,Z 66.500,A 180.000,B 0.000,C 180.000} C_DIS
LIN {X 112.479,Y 96.718,Z 66.500,A 180.000,B 0.000,C 180.000} C_DIS
LIN {X 112.467,Y 96.539,Z 66.500,A 180.000,B 0.000,C 180.000} C_DIS
LIN {X 112.422,Y 96.003,Z 66.500,A 180.000,B 0.000,C 180.000} C_DIS
LIN {X 112.406,Y 95.824,Z 66.500,A 180.000,B 0.000,C 180.000} C_DIS
LIN {X 112.382,Y 95.645,Z 66.500,A 180.000,B 0.000,C 180.000} C_DIS
LIN {X 112.306,Y 95.109,Z 66.500,A 180.000,B 0.000,C 180.000} C_DIS
LIN {X 112.278,Y 94.930,Z 66.500,A 180.000,B 0.000,C 180.000} C_DIS
LIN {X 112.271,Y 94.895,Z 66.500,A 180.000,B 0.000,C 180.000} C_DIS
LIN {X 112.171,Y 94.394,Z 66.500,A 180.000,B 0.000,C 180.000} C_DIS
LIN {X 112.135,Y 94.215,Z 66.500,A 180.000,B 0.000,C 180.000} C_DIS
LIN {X 112.092,Y 94.036,Z 66.500,A 180.000,B 0.000,C 180.000} C_DIS
LIN {X 111.954,Y 93.500,Z 66.500,A 180.000,B 0.000,C 180.000} C_DIS
LIN {X 111.913,Y 93.346,Z 66.500,A 180.000,B 0.000,C 180.000} C_DIS
LIN {X 111.906,Y 93.321,Z 66.500,A 180.000,B 0.000,C 180.000} C_DIS
LIN {X 111.849,Y 93.142,Z 66.500,A 180.000,B 0.000,C 180.000} C_DIS
LIN {X 111.734,Y 92.782,Z 66.500,A 180.000,B 0.000,C 180.000} C_DIS
LIN {X 111.678,Y 92.606,Z 66.500,A 180.000,B 0.000,C 180.000} C_DIS
LIN {X 111.614,Y 92.427,Z 66.500,A 180.000,B 0.000,C 180.000} C_DIS
LIN {X 111.409,Y 91.891,Z 66.500,A 180.000,B 0.000,C 180.000} C_DIS
LIN {X 111.377,Y 91.806,Z 66.500,A 180.000,B 0.000,C 180.000} C_DIS
LIN {X 111.338,Y 91.712,Z 66.500,A 180.000,B 0.000,C 180.000} C_DIS
LIN {X 111.258,Y 91.533,Z 66.500,A 180.000,B 0.000,C 180.000} C_DIS
LIN {X 111.098,Y 91.176,Z 66.500,A 180.000,B 0.000,C 180.000} C_DIS
LIN {X 111.019,Y 91.002,Z 66.500,A 180.000,B 0.000,C 180.000} C_DIS
LIN {X 111.017,Y 90.997,Z 66.500,A 180.000,B 0.000,C 180.000} C_DIS
LIN {X 110.926,Y 90.818,Z 66.500,A 180.000,B 0.000,C 180.000} C_DIS
LIN {X 110.662,Y 90.307,Z 66.500,A 180.000,B 0.000,C 180.000} C_DIS
LIN {X 110.649,Y 90.282,Z 66.500,A 180.000,B 0.000,C 180.000} C_DIS
LIN {X 110.546,Y 90.103,Z 66.500,A 180.000,B 0.000,C 180.000} C_DIS
LIN {X 110.304,Y 89.693,Z 66.500,A 180.000,B 0.000,C 180.000} C_DIS
LIN {X 110.230,Y 89.567,Z 66.500,A 180.000,B 0.000,C 180.000} C_DIS
LIN {X 110.126,Y 89.405,Z 66.500,A 180.000,B 0.000,C 180.000} C_DIS
LIN {X 109.875,Y 89.031,Z 66.500,A 180.000,B 0.000,C 180.000} C_DIS
LIN {X 109.768,Y 88.870,Z 66.500,A 180.000,B 0.000,C 180.000} C_DIS
LIN {X 109.756,Y 88.852,Z 66.500,A 180.000,B 0.000,C 180.000} C_DIS
LIN {X 109.624,Y 88.673,Z 66.500,A 180.000,B 0.000,C 180.000} C_DIS
LIN {X 109.355,Y 88.316,Z 66.500,A 180.000,B 0.000,C 180.000} C_DIS
LIN {X 109.232,Y 88.153,Z 66.500,A 180.000,B 0.000,C 180.000} C_DIS
LIN {X 109.219,Y 88.137,Z 66.500,A 180.000,B 0.000,C 180.000} C_DIS
LIN {X 109.069,Y 87.958,Z 66.500,A 180.000,B 0.000,C 180.000} C_DIS
LIN {X 108.767,Y 87.601,Z 66.500,A 180.000,B 0.000,C 180.000} C_DIS
LIN {X 108.695,Y 87.517,Z 66.500,A 180.000,B 0.000,C 180.000} C_DIS
LIN {X 108.607,Y 87.422,Z 66.500,A 180.000,B 0.000,C 180.000} C_DIS
LIN {X 108.159,Y 86.947,Z 66.500,A 180.000,B 0.000,C 180.000} C_DIS
LIN {X 108.099,Y 86.885,Z 66.500,A 180.000,B 0.000,C 180.000} C_DIS
LIN {X 107.980,Y 86.773,Z 66.500,A 180.000,B 0.000,C 180.000} C_DIS
LIN {X 107.623,Y 86.435,Z 66.500,A 180.000,B 0.000,C 180.000} C_DIS
LIN {X 107.532,Y 86.349,Z 66.500,A 180.000,B 0.000,C 180.000} C_DIS
LIN {X 107.444,Y 86.271,Z 66.500,A 180.000,B 0.000,C 180.000} C_DIS
LIN {X 106.908,Y 85.818,Z 66.500,A 180.000,B 0.000,C 180.000} C_DIS
LIN {X 106.902,Y 85.813,Z 66.500,A 180.000,B 0.000,C 180.000} C_DIS
LIN {X 106.729,Y 85.678,Z 66.500,A 180.000,B 0.000,C 180.000} C_DIS
LIN {X 106.371,Y 85.409,Z 66.500,A 180.000,B 0.000,C 180.000} C_DIS
LIN {X 106.194,Y 85.276,Z 66.500,A 180.000,B 0.000,C 180.000} C_DIS
LIN {X 106.193,Y 85.276,Z 66.500,A 180.000,B 0.000,C 180.000} C_DIS
LIN {X 106.014,Y 85.154,Z 66.500,A 180.000,B 0.000,C 180.000} C_DIS
LIN {X 105.656,Y 84.915,Z 66.500,A 180.000,B 0.000,C 180.000} C_DIS
LIN {X 105.477,Y 84.797,Z 66.500,A 180.000,B 0.000,C 180.000} C_DIS
LIN {X 105.382,Y 84.740,Z 66.500,A 180.000,B 0.000,C 180.000} C_DIS
LIN {X 104.941,Y 84.480,Z 66.500,A 180.000,B 0.000,C 180.000} C_DIS
LIN {X 104.775,Y 84.383,Z 66.500,A 180.000,B 0.000,C 180.000} C_DIS
LIN {X 104.762,Y 84.375,Z 66.500,A 180.000,B 0.000,C 180.000} C_DIS
LIN {X 104.584,Y 84.282,Z 66.500,A 180.000,B 0.000,C 180.000} C_DIS
LIN {X 104.087,Y 84.025,Z 66.500,A 180.000,B 0.000,C 180.000} C_DIS
LIN {X 104.047,Y 84.005,Z 66.500,A 180.000,B 0.000,C 180.000} C_DIS
LIN {X 103.869,Y 83.922,Z 66.500,A 180.000,B 0.000,C 180.000} C_DIS
LIN {X 103.300,Y 83.668,Z 66.500,A 180.000,B 0.000,C 180.000} C_DIS
LIN {X 103.153,Y 83.608,Z 66.500,A 180.000,B 0.000,C 180.000} C_DIS
LIN {X 102.617,Y 83.403,Z 66.500,A 180.000,B 0.000,C 180.000} C_DIS
LIN {X 102.438,Y 83.336,Z 66.500,A 180.000,B 0.000,C 180.000} C_DIS
LIN {X 102.358,Y 83.310,Z 66.500,A 180.000,B 0.000,C 180.000} C_DIS
LIN {X 101.723,Y 83.108,Z 66.500,A 180.000,B 0.000,C 180.000} C_DIS
LIN {X 101.545,Y 83.057,Z 66.500,A 180.000,B 0.000,C 180.000} C_DIS
LIN {X 101.008,Y 82.919,Z 66.500,A 180.000,B 0.000,C 180.000} C_DIS
LIN {X 100.829,Y 82.874,Z 66.500,A 180.000,B 0.000,C 180.000} C_DIS
LIN {X 100.651,Y 82.838,Z 66.500,A 180.000,B 0.000,C 180.000} C_DIS
LIN {X 100.114,Y 82.731,Z 66.500,A 180.000,B 0.000,C 180.000} C_DIS
LIN {X 99.936,Y 82.700,Z 66.500,A 180.000,B 0.000,C 180.000} C_DIS
LIN {X 99.399,Y 82.624,Z 66.500,A 180.000,B 0.000,C 180.000} C_DIS
LIN {X 99.221,Y 82.599,Z 66.500,A 180.000,B 0.000,C 180.000} C_DIS
LIN {X 99.185,Y 82.595,Z 66.500,A 180.000,B 0.000,C 180.000} C_DIS
LIN {X 99.042,Y 82.582,Z 66.500,A 180.000,B 0.000,C 180.000} C_DIS
LIN {X 98.505,Y 82.536,Z 66.500,A 180.000,B 0.000,C 180.000} C_DIS
LIN {X 98.327,Y 82.523,Z 66.500,A 180.000,B 0.000,C 180.000} C_DIS
LIN {X 98.148,Y 82.517,Z 66.500,A 180.000,B 0.000,C 180.000} C_DIS
LIN {X 97.612,Y 82.502,Z 66.500,A 180.000,B 0.000,C 180.000} C_DIS
LIN {X 97.433,Y 82.501,Z 66.500,A 180.000,B 0.000,C 180.000} C_DIS
LIN {X 96.897,Y 82.516,Z 66.500,A 180.000,B 0.000,C 180.000} C_DIS
LIN {X 96.718,Y 82.521,Z 66.500,A 180.000,B 0.000,C 180.000} C_DIS
LIN {X 96.539,Y 82.533,Z 66.500,A 180.000,B 0.000,C 180.000} C_DIS
LIN {X 96.003,Y 82.578,Z 66.500,A 180.000,B 0.000,C 180.000} C_DIS
LIN {X 95.824,Y 82.594,Z 66.500,A 180.000,B 0.000,C 180.000} C_DIS
LIN {X 95.815,Y 82.595,Z 66.500,A 180.000,B 0.000,C 180.000} C_DIS
LIN {X 95.645,Y 82.618,Z 66.500,A 180.000,B 0.000,C 180.000} C_DIS
LIN {X 95.109,Y 82.694,Z 66.500,A 180.000,B 0.000,C 180.000} C_DIS
LIN {X 94.930,Y 82.722,Z 66.500,A 180.000,B 0.000,C 180.000} C_DIS
LIN {X 94.751,Y 82.758,Z 66.500,A 180.000,B 0.000,C 180.000} C_DIS
LIN {X 94.394,Y 82.829,Z 66.500,A 180.000,B 0.000,C 180.000} C_DIS
LIN {X 94.215,Y 82.865,Z 66.500,A 180.000,B 0.000,C 180.000} C_DIS
LIN {X 94.036,Y 82.908,Z 66.500,A 180.000,B 0.000,C 180.000} C_DIS
LIN {X 93.500,Y 83.046,Z 66.500,A 180.000,B 0.000,C 180.000} C_DIS
LIN {X 93.321,Y 83.094,Z 66.500,A 180.000,B 0.000,C 180.000} C_DIS
LIN {X 93.203,Y 83.131,Z 66.500,A 180.000,B 0.000,C 180.000} C_DIS
LIN {X 92.642,Y 83.310,Z 66.500,A 180.000,B 0.000,C 180.000} C_DIS
LIN {X 92.606,Y 83.322,Z 66.500,A 180.000,B 0.000,C 180.000} C_DIS
LIN {X 92.427,Y 83.386,Z 66.500,A 180.000,B 0.000,C 180.000} C_DIS
LIN {X 91.891,Y 83.591,Z 66.500,A 180.000,B 0.000,C 180.000} C_DIS
LIN {X 91.712,Y 83.662,Z 66.500,A 180.000,B 0.000,C 180.000} C_DIS
LIN {X 91.700,Y 83.668,Z 66.500,A 180.000,B 0.000,C 180.000} C_DIS
LIN {X 91.176,Y 83.902,Z 66.500,A 180.000,B 0.000,C 180.000} C_DIS
LIN {X 90.997,Y 83.983,Z 66.500,A 180.000,B 0.000,C 180.000} C_DIS
LIN {X 90.913,Y 84.025,Z 66.500,A 180.000,B 0.000,C 180.000} C_DIS
LIN {X 90.461,Y 84.259,Z 66.500,A 180.000,B 0.000,C 180.000} C_DIS
LIN {X 90.282,Y 84.351,Z 66.500,A 180.000,B 0.000,C 180.000} C_DIS
LIN {X 90.225,Y 84.383,Z 66.500,A 180.000,B 0.000,C 180.000} C_DIS
LIN {X 90.103,Y 84.454,Z 66.500,A 180.000,B 0.000,C 180.000} C_DIS
LIN {X 89.618,Y 84.740,Z 66.500,A 180.000,B 0.000,C 180.000} C_DIS
LIN {X 89.567,Y 84.770,Z 66.500,A 180.000,B 0.000,C 180.000} C_DIS
LIN {X 89.388,Y 84.886,Z 66.500,A 180.000,B 0.000,C 180.000} C_DIS
LIN {X 89.031,Y 85.125,Z 66.500,A 180.000,B 0.000,C 180.000} C_DIS
LIN {X 88.852,Y 85.244,Z 66.500,A 180.000,B 0.000,C 180.000} C_DIS
LIN {X 88.806,Y 85.276,Z 66.500,A 180.000,B 0.000,C 180.000} C_DIS
LIN {X 88.673,Y 85.376,Z 66.500,A 180.000,B 0.000,C 180.000} C_DIS
LIN {X 88.316,Y 85.645,Z 66.500,A 180.000,B 0.000,C 180.000} C_DIS
LIN {X 88.137,Y 85.781,Z 66.500,A 180.000,B 0.000,C 180.000} C_DIS
LIN {X 88.098,Y 85.813,Z 66.500,A 180.000,B 0.000,C 180.000} C_DIS
LIN {X 87.779,Y 86.082,Z 66.500,A 180.000,B 0.000,C 180.000} C_DIS
LIN {X 87.601,Y 86.233,Z 66.500,A 180.000,B 0.000,C 180.000} C_DIS
LIN {X 87.468,Y 86.349,Z 66.500,A 180.000,B 0.000,C 180.000} C_DIS
LIN {X 87.422,Y 86.393,Z 66.500,A 180.000,B 0.000,C 180.000} C_DIS
LIN {X 87.064,Y 86.731,Z 66.500,A 180.000,B 0.000,C 180.000} C_DIS
LIN {X 86.901,Y 86.885,Z 66.500,A 180.000,B 0.000,C 180.000} C_DIS
LIN {X 86.885,Y 86.901,Z 66.500,A 180.000,B 0.000,C 180.000} C_DIS
LIN {X 86.731,Y 87.064,Z 66.500,A 180.000,B 0.000,C 180.000} C_DIS
LIN {X 86.393,Y 87.422,Z 66.500,A 180.000,B 0.000,C 180.000} C_DIS
LIN {X 86.349,Y 87.468,Z 66.500,A 180.000,B 0.000,C 180.000} C_DIS
LIN {X 86.233,Y 87.601,Z 66.500,A 180.000,B 0.000,C 180.000} C_DIS
LIN {X 85.931,Y 87.958,Z 66.500,A 180.000,B 0.000,C 180.000} C_DIS
LIN {X 85.813,Y 88.098,Z 66.500,A 180.000,B 0.000,C 180.000} C_DIS
LIN {X 85.781,Y 88.137,Z 66.500,A 180.000,B 0.000,C 180.000} C_DIS
LIN {X 85.645,Y 88.316,Z 66.500,A 180.000,B 0.000,C 180.000} C_DIS
LIN {X 85.376,Y 88.673,Z 66.500,A 180.000,B 0.000,C 180.000} C_DIS
LIN {X 85.276,Y 88.806,Z 66.500,A 180.000,B 0.000,C 180.000} C_DIS
LIN {X 85.244,Y 88.852,Z 66.500,A 180.000,B 0.000,C 180.000} C_DIS
LIN {X 85.125,Y 89.031,Z 66.500,A 180.000,B 0.000,C 180.000} C_DIS
LIN {X 84.886,Y 89.388,Z 66.500,A 180.000,B 0.000,C 180.000} C_DIS
LIN {X 84.770,Y 89.567,Z 66.500,A 180.000,B 0.000,C 180.000} C_DIS
LIN {X 84.740,Y 89.618,Z 66.500,A 180.000,B 0.000,C 180.000} C_DIS
LIN {X 84.454,Y 90.103,Z 66.500,A 180.000,B 0.000,C 180.000} C_DIS
LIN {X 84.383,Y 90.225,Z 66.500,A 180.000,B 0.000,C 180.000} C_DIS
LIN {X 84.351,Y 90.282,Z 66.500,A 180.000,B 0.000,C 180.000} C_DIS
LIN {X 84.259,Y 90.461,Z 66.500,A 180.000,B 0.000,C 180.000} C_DIS
LIN {X 84.025,Y 90.913,Z 66.500,A 180.000,B 0.000,C 180.000} C_DIS
LIN {X 83.983,Y 90.997,Z 66.500,A 180.000,B 0.000,C 180.000} C_DIS
LIN {X 83.902,Y 91.176,Z 66.500,A 180.000,B 0.000,C 180.000} C_DIS
LIN {X 83.668,Y 91.700,Z 66.500,A 180.000,B 0.000,C 180.000} C_DIS
LIN {X 83.662,Y 91.712,Z 66.500,A 180.000,B 0.000,C 180.000} C_DIS
LIN {X 83.591,Y 91.891,Z 66.500,A 180.000,B 0.000,C 180.000} C_DIS
LIN {X 83.386,Y 92.427,Z 66.500,A 180.000,B 0.000,C 180.000} C_DIS
LIN {X 83.322,Y 92.606,Z 66.500,A 180.000,B 0.000,C 180.000} C_DIS
LIN {X 83.310,Y 92.642,Z 66.500,A 180.000,B 0.000,C 180.000} C_DIS
LIN {X 83.131,Y 93.203,Z 66.500,A 180.000,B 0.000,C 180.000} C_DIS
LIN {X 83.094,Y 93.321,Z 66.500,A 180.000,B 0.000,C 180.000} C_DIS
LIN {X 83.046,Y 93.500,Z 66.500,A 180.000,B 0.000,C 180.000} C_DIS
LIN {X 82.908,Y 94.036,Z 66.500,A 180.000,B 0.000,C 180.000} C_DIS
LIN {X 82.865,Y 94.215,Z 66.500,A 180.000,B 0.000,C 180.000} C_DIS
LIN {X 82.829,Y 94.394,Z 66.500,A 180.000,B 0.000,C 180.000} C_DIS
LIN {X 82.758,Y 94.751,Z 66.500,A 180.000,B 0.000,C 180.000} C_DIS
LIN {X 82.722,Y 94.930,Z 66.500,A 180.000,B 0.000,C 180.000} C_DIS
LIN {X 82.694,Y 95.109,Z 66.500,A 180.000,B 0.000,C 180.000} C_DIS
LIN {X 82.618,Y 95.645,Z 66.500,A 180.000,B 0.000,C 180.000} C_DIS
LIN {X 82.595,Y 95.815,Z 66.500,A 180.000,B 0.000,C 180.000} C_DIS
LIN {X 82.594,Y 95.824,Z 66.500,A 180.000,B 0.000,C 180.000} C_DIS
LIN {X 82.578,Y 96.003,Z 66.500,A 180.000,B 0.000,C 180.000} C_DIS
LIN {X 82.533,Y 96.539,Z 66.500,A 180.000,B 0.000,C 180.000} C_DIS
LIN {X 82.521,Y 96.718,Z 66.500,A 180.000,B 0.000,C 180.000} C_DIS
LIN {X 82.516,Y 96.897,Z 66.500,A 180.000,B 0.000,C 180.000} C_DIS
LIN {X 82.501,Y 97.433,Z 66.500,A 180.000,B 0.000,C 180.000} C_DIS
LIN {X 82.502,Y 97.612,Z 66.500,A 180.000,B 0.000,C 180.000} C_DIS
LIN {X 82.517,Y 98.148,Z 66.500,A 180.000,B 0.000,C 180.000} C_DIS
LIN {X 82.523,Y 98.327,Z 66.500,A 180.000,B 0.000,C 180.000} C_DIS
LIN {X 82.536,Y 98.505,Z 66.500,A 180.000,B 0.000,C 180.000} C_DIS
LIN {X 82.582,Y 99.042,Z 66.500,A 180.000,B 0.000,C 180.000} C_DIS
LIN {X 82.595,Y 99.185,Z 66.500,A 180.000,B 0.000,C 180.000} C_DIS
LIN {X 82.599,Y 99.221,Z 66.500,A 180.000,B 0.000,C 180.000} C_DIS
LIN {X 82.624,Y 99.399,Z 66.500,A 180.000,B 0.000,C 180.000} C_DIS
LIN {X 82.700,Y 99.936,Z 66.500,A 180.000,B 0.000,C 180.000} C_DIS
LIN {X 82.731,Y 100.114,Z 66.500,A 180.000,B 0.000,C 180.000} C_DIS
LIN {X 82.838,Y 100.651,Z 66.500,A 180.000,B 0.000,C 180.000} C_DIS
LIN {X 82.874,Y 100.829,Z 66.500,A 180.000,B 0.000,C 180.000} C_DIS
LIN {X 82.919,Y 101.008,Z 66.500,A 180.000,B 0.000,C 180.000} C_DIS
LIN {X 83.057,Y 101.545,Z 66.500,A 180.000,B 0.000,C 180.000} C_DIS
LIN {X 83.108,Y 101.723,Z 66.500,A 180.000,B 0.000,C 180.000} C_DIS
LIN {X 83.310,Y 102.358,Z 66.500,A 180.000,B 0.000,C 180.000} C_DIS
LIN {X 83.336,Y 102.438,Z 66.500,A 180.000,B 0.000,C 180.000} C_DIS
LIN {X 83.403,Y 102.617,Z 66.500,A 180.000,B 0.000,C 180.000} C_DIS
LIN {X 83.608,Y 103.153,Z 66.500,A 180.000,B 0.000,C 180.000} C_DIS
LIN {X 83.668,Y 103.300,Z 66.500,A 180.000,B 0.000,C 180.000} C_DIS
LIN {X 83.922,Y 103.869,Z 66.500,A 180.000,B 0.000,C 180.000} C_DIS
LIN {X 84.005,Y 104.047,Z 66.500,A 180.000,B 0.000,C 180.000} C_DIS
LIN {X 84.025,Y 104.087,Z 66.500,A 180.000,B 0.000,C 180.000} C_DIS
LIN {X 84.282,Y 104.584,Z 66.500,A 180.000,B 0.000,C 180.000} C_DIS
LIN {X 84.375,Y 104.762,Z 66.500,A 180.000,B 0.000,C 180.000} C_DIS
LIN {X 84.383,Y 104.775,Z 66.500,A 180.000,B 0.000,C 180.000} C_DIS
LIN {X 84.480,Y 104.941,Z 66.500,A 180.000,B 0.000,C 180.000} C_DIS
LIN {X 84.740,Y 105.382,Z 66.500,A 180.000,B 0.000,C 180.000} C_DIS
LIN {X 84.797,Y 105.477,Z 66.500,A 180.000,B 0.000,C 180.000} C_DIS
LIN {X 84.915,Y 105.656,Z 66.500,A 180.000,B 0.000,C 180.000} C_DIS
LIN {X 85.154,Y 106.014,Z 66.500,A 180.000,B 0.000,C 180.000} C_DIS
LIN {X 85.276,Y 106.193,Z 66.500,A 180.000,B 0.000,C 180.000} C_DIS
LIN {X 85.276,Y 106.194,Z 66.500,A 180.000,B 0.000,C 180.000} C_DIS
LIN {X 85.409,Y 106.371,Z 66.500,A 180.000,B 0.000,C 180.000} C_DIS
LIN {X 85.678,Y 106.729,Z 66.500,A 180.000,B 0.000,C 180.000} C_DIS
LIN {X 85.813,Y 106.902,Z 66.500,A 180.000,B 0.000,C 180.000} C_DIS
LIN {X 85.818,Y 106.908,Z 66.500,A 180.000,B 0.000,C 180.000} C_DIS
LIN {X 86.271,Y 107.444,Z 66.500,A 180.000,B 0.000,C 180.000} C_DIS
LIN {X 86.349,Y 107.532,Z 66.500,A 180.000,B 0.000,C 180.000} C_DIS
LIN {X 86.435,Y 107.623,Z 66.500,A 180.000,B 0.000,C 180.000} C_DIS
LIN {X 86.773,Y 107.980,Z 66.500,A 180.000,B 0.000,C 180.000} C_DIS
LIN {X 86.885,Y 108.099,Z 66.500,A 180.000,B 0.000,C 180.000} C_DIS
LIN {X 86.947,Y 108.159,Z 66.500,A 180.000,B 0.000,C 180.000} C_DIS
LIN {X 87.422,Y 108.607,Z 66.500,A 180.000,B 0.000,C 180.000} C_DIS
LIN {X 87.517,Y 108.695,Z 66.500,A 180.000,B 0.000,C 180.000} C_DIS
LIN {X 87.601,Y 108.767,Z 66.500,A 180.000,B 0.000,C 180.000} C_DIS
LIN {X 87.958,Y 109.069,Z 66.500,A 180.000,B 0.000,C 180.000} C_DIS
LIN {X 88.137,Y 109.219,Z 66.500,A 180.000,B 0.000,C 180.000} C_DIS
LIN {X 88.153,Y 109.232,Z 66.500,A 180.000,B 0.000,C 180.000} C_DIS
LIN {X 88.316,Y 109.355,Z 66.500,A 180.000,B 0.000,C 180.000} C_DIS
LIN {X 88.673,Y 109.624,Z 66.500,A 180.000,B 0.000,C 180.000} C_DIS
LIN {X 88.852,Y 109.756,Z 66.500,A 180.000,B 0.000,C 180.000} C_DIS
LIN {X 88.870,Y 109.768,Z 66.500,A 180.000,B 0.000,C 180.000} C_DIS
LIN {X 89.031,Y 109.875,Z 66.500,A 180.000,B 0.000,C 180.000} C_DIS
LIN {X 89.405,Y 110.126,Z 66.500,A 180.000,B 0.000,C 180.000} C_DIS
LIN {X 89.567,Y 110.230,Z 66.500,A 180.000,B 0.000,C 180.000} C_DIS
LIN {X 89.693,Y 110.304,Z 66.500,A 180.000,B 0.000,C 180.000} C_DIS
LIN {X 90.103,Y 110.546,Z 66.500,A 180.000,B 0.000,C 180.000} C_DIS
LIN {X 90.282,Y 110.649,Z 66.500,A 180.000,B 0.000,C 180.000} C_DIS
LIN {X 90.307,Y 110.662,Z 66.500,A 180.000,B 0.000,C 180.000} C_DIS
LIN {X 90.818,Y 110.926,Z 66.500,A 180.000,B 0.000,C 180.000} C_DIS
LIN {X 90.997,Y 111.017,Z 66.500,A 180.000,B 0.000,C 180.000} C_DIS
LIN {X 91.002,Y 111.019,Z 66.500,A 180.000,B 0.000,C 180.000} C_DIS
LIN {X 91.070,Y 111.050,Z 66.500,A 180.000,B 0.000,C 180.000} C_DIS
; Link Move Starts
LIN {X 91.357,Y 111.179,Z 66.500,A 180.000,B 0.000,C 180.000} C_DIS
LIN {X 91.644,Y 111.308,Z 66.499,A 180.000,B 0.000,C 180.000} C_DIS
LIN {X 91.936,Y 111.427,Z 66.498,A 180.000,B 0.000,C 180.000} C_DIS
LIN {X 92.230,Y 111.539,Z 66.496,A 180.000,B 0.000,C 180.000} C_DIS
LIN {X 92.525,Y 111.651,Z 66.494,A 180.000,B 0.000,C 180.000} C_DIS
LIN {X 92.824,Y 111.748,Z 66.491,A 180.000,B 0.000,C 180.000} C_DIS
LIN {X 93.124,Y 111.844,Z 66.488,A 180.000,B 0.000,C 180.000} C_DIS
LIN {X 93.426,Y 111.935,Z 66.485,A 180.000,B 0.000,C 180.000} C_DIS
LIN {X 93.731,Y 112.014,Z 66.481,A 180.000,B 0.000,C 180.000} C_DIS
LIN {X 94.036,Y 112.092,Z 66.477,A 180.000,B 0.000,C 180.000} C_DIS
LIN {X 94.343,Y 112.161,Z 66.472,A 180.000,B 0.000,C 180.000} C_DIS
LIN {X 94.498,Y 112.192,Z 66.469,A 180.000,B 0.000,C 180.000} C_DIS
LIN {X 94.652,Y 112.222,Z 66.467,A 180.000,B 0.000,C 180.000} C_DIS
LIN {X 94.807,Y 112.253,Z 66.464,A 180.000,B 0.000,C 180.000} C_DIS
LIN {X 94.961,Y 112.283,Z 66.461,A 180.000,B 0.000,C 180.000} C_DIS
LIN {X 95.117,Y 112.307,Z 66.459,A 180.000,B 0.000,C 180.000} C_DIS
LIN {X 95.273,Y 112.329,Z 66.456,A 180.000,B 0.000,C 180.000} C_DIS
LIN {X 95.429,Y 112.351,Z 66.452,A 180.000,B 0.000,C 180.000} C_DIS
LIN {X 95.585,Y 112.373,Z 66.449,A 180.000,B 0.000,C 180.000} C_DIS
LIN {X 95.741,Y 112.395,Z 66.446,A 180.000,B 0.000,C 180.000} C_DIS
LIN {X 95.897,Y 112.413,Z 66.443,A 180.000,B 0.000,C 180.000} C_DIS
LIN {X 96.054,Y 112.426,Z 66.439,A 180.000,B 0.000,C 180.000} C_DIS
LIN {X 96.211,Y 112.440,Z 66.436,A 180.000,B 0.000,C 180.000} C_DIS
LIN {X 96.368,Y 112.453,Z 66.432,A 180.000,B 0.000,C 180.000} C_DIS
LIN {X 96.525,Y 112.466,Z 66.428,A 180.000,B 0.000,C 180.000} C_DIS
LIN {X 96.682,Y 112.478,Z 66.425,A 180.000,B 0.000,C 180.000} C_DIS
LIN {X 96.840,Y 112.482,Z 66.421,A 180.000,B 0.000,C 180.000} C_DIS
LIN {X 96.997,Y 112.487,Z 66.417,A 180.000,B 0.000,C 180.000} C_DIS
LIN {X 97.154,Y 112.491,Z 66.413,A 180.000,B 0.000,C 180.000} C_DIS
LIN {X 97.312,Y 112.496,Z 66.409,A 180.000,B 0.000,C 180.000} C_DIS
LIN {X 97.469,Y 112.500,Z 66.405,A 180.000,B 0.000,C 180.000} C_DIS
LIN {X 97.627,Y 112.497,Z 66.400,A 180.000,B 0.000,C 180.000} C_DIS
LIN {X 97.784,Y 112.493,Z 66.396,A 180.000,B 0.000,C 180.000} C_DIS
LIN {X 97.942,Y 112.489,Z 66.392,A 180.000,B 0.000,C 180.000} C_DIS
LIN {X 98.099,Y 112.484,Z 66.387,A 180.000,B 0.000,C 180.000} C_DIS
LIN {X 98.257,Y 112.480,Z 66.383,A 180.000,B 0.000,C 180.000} C_DIS
LIN {X 98.414,Y 112.471,Z 66.378,A 180.000,B 0.000,C 180.000} C_DIS
LIN {X 98.571,Y 112.458,Z 66.373,A 180.000,B 0.000,C 180.000} C_DIS
LIN {X 98.728,Y 112.445,Z 66.369,A 180.000,B 0.000,C 180.000} C_DIS
LIN {X 98.885,Y 112.432,Z 66.364,A 180.000,B 0.000,C 180.000} C_DIS
LIN {X 99.042,Y 112.418,Z 66.359,A 180.000,B 0.000,C 180.000} C_DIS
LIN {X 99.198,Y 112.403,Z 66.354,A 180.000,B 0.000,C 180.000} C_DIS
LIN {X 99.276,Y 112.393,Z 66.351,A 180.000,B 0.000,C 180.000} C_DIS
LIN {X 99.354,Y 112.382,Z 66.349,A 180.000,B 0.000,C 180.000} C_DIS
LIN {X 99.432,Y 112.371,Z 66.346,A 180.000,B 0.000,C 180.000} C_DIS
LIN {X 99.510,Y 112.360,Z 66.344,A 180.000,B 0.000,C 180.000} C_DIS
LIN {X 99.588,Y 112.349,Z 66.341,A 180.000,B 0.000,C 180.000} C_DIS
LIN {X 99.666,Y 112.338,Z 66.339,A 180.000,B 0.000,C 180.000} C_DIS
LIN {X 99.744,Y 112.327,Z 66.336,A 180.000,B 0.000,C 180.000} C_DIS
LIN {X 99.900,Y 112.305,Z 66.331,A 180.000,B 0.000,C 180.000} C_DIS
LIN {X 99.978,Y 112.294,Z 66.328,A 180.000,B 0.000,C 180.000} C_DIS
LIN {X 100.056,Y 112.280,Z 66.325,A 180.000,B 0.000,C 180.000} C_DIS
LIN {X 100.133,Y 112.265,Z 66.323,A 180.000,B 0.000,C 180.000} C_DIS
LIN {X 100.288,Y 112.234,Z 66.317,A 180.000,B 0.000,C 180.000} C_DIS
LIN {X 100.442,Y 112.204,Z 66.312,A 180.000,B 0.000,C 180.000} C_DIS
LIN {X 100.751,Y 112.142,Z 66.301,A 180.000,B 0.000,C 180.000} C_DIS
LIN {X 100.828,Y 112.126,Z 66.298,A 180.000,B 0.000,C 180.000} C_DIS
LIN {X 100.905,Y 112.108,Z 66.296,A 180.000,B 0.000,C 180.000} C_DIS
LIN {X 101.057,Y 112.068,Z 66.290,A 180.000,B 0.000,C 180.000} C_DIS
LIN {X 101.286,Y 112.009,Z 66.282,A 180.000,B 0.000,C 180.000} C_DIS
LIN {X 101.438,Y 111.970,Z 66.276,A 180.000,B 0.000,C 180.000} C_DIS
LIN {X 101.515,Y 111.950,Z 66.274,A 180.000,B 0.000,C 180.000} C_DIS
LIN {X 101.591,Y 111.931,Z 66.271,A 180.000,B 0.000,C 180.000} C_DIS
LIN {X 101.667,Y 111.910,Z 66.268,A 180.000,B 0.000,C 180.000} C_DIS
LIN {X 101.742,Y 111.886,Z 66.265,A 180.000,B 0.000,C 180.000} C_DIS
LIN {X 101.817,Y 111.862,Z 66.263,A 180.000,B 0.000,C 180.000} C_DIS
LIN {X 101.967,Y 111.815,Z 66.257,A 180.000,B 0.000,C 180.000} C_DIS
LIN {X 102.192,Y 111.743,Z 66.249,A 180.000,B 0.000,C 180.000} C_DIS
LIN {X 102.342,Y 111.695,Z 66.243,A 180.000,B 0.000,C 180.000} C_DIS
LIN {X 102.417,Y 111.671,Z 66.241,A 180.000,B 0.000,C 180.000} C_DIS
LIN {X 102.492,Y 111.645,Z 66.238,A 180.000,B 0.000,C 180.000} C_DIS
LIN {X 102.565,Y 111.617,Z 66.235,A 180.000,B 0.000,C 180.000} C_DIS
LIN {X 102.786,Y 111.533,Z 66.227,A 180.000,B 0.000,C 180.000} C_DIS
LIN {X 102.933,Y 111.476,Z 66.221,A 180.000,B 0.000,C 180.000} C_DIS
LIN {X 103.007,Y 111.448,Z 66.219,A 180.000,B 0.000,C 180.000} C_DIS
LIN {X 103.154,Y 111.392,Z 66.213,A 180.000,B 0.000,C 180.000} C_DIS
LIN {X 103.227,Y 111.364,Z 66.210,A 180.000,B 0.000,C 180.000} C_DIS
LIN {X 103.300,Y 111.333,Z 66.208,A 180.000,B 0.000,C 180.000} C_DIS
LIN {X 103.443,Y 111.268,Z 66.202,A 180.000,B 0.000,C 180.000} C_DIS
LIN {X 103.875,Y 111.075,Z 66.186,A 180.000,B 0.000,C 180.000} C_DIS
LIN {X 103.947,Y 111.043,Z 66.183,A 180.000,B 0.000,C 180.000} C_DIS
LIN {X 104.018,Y 111.010,Z 66.180,A 180.000,B 0.000,C 180.000} C_DIS
LIN {X 104.088,Y 110.974,Z 66.177,A 180.000,B 0.000,C 180.000} C_DIS
LIN {X 104.158,Y 110.938,Z 66.175,A 180.000,B 0.000,C 180.000} C_DIS
LIN {X 104.298,Y 110.866,Z 66.169,A 180.000,B 0.000,C 180.000} C_DIS
LIN {X 104.648,Y 110.685,Z 66.155,A 180.000,B 0.000,C 180.000} C_DIS
LIN {X 104.718,Y 110.649,Z 66.153,A 180.000,B 0.000,C 180.000} C_DIS
LIN {X 104.787,Y 110.611,Z 66.150,A 180.000,B 0.000,C 180.000} C_DIS
LIN {X 104.855,Y 110.571,Z 66.147,A 180.000,B 0.000,C 180.000} C_DIS
LIN {X 105.330,Y 110.291,Z 66.128,A 180.000,B 0.000,C 180.000} C_DIS
LIN {X 105.397,Y 110.251,Z 66.125,A 180.000,B 0.000,C 180.000} C_DIS
LIN {X 105.465,Y 110.211,Z 66.122,A 180.000,B 0.000,C 180.000} C_DIS
LIN {X 105.531,Y 110.168,Z 66.120,A 180.000,B 0.000,C 180.000} C_DIS
LIN {X 105.597,Y 110.124,Z 66.117,A 180.000,B 0.000,C 180.000} C_DIS
LIN {X 105.990,Y 109.862,Z 66.100,A 180.000,B 0.000,C 180.000} C_DIS
LIN {X 106.121,Y 109.774,Z 66.095,A 180.000,B 0.000,C 180.000} C_DIS
LIN {X 106.185,Y 109.730,Z 66.092,A 180.000,B 0.000,C 180.000} C_DIS
LIN {X 106.249,Y 109.683,Z 66.089,A 180.000,B 0.000,C 180.000} C_DIS
LIN {X 106.563,Y 109.446,Z 66.076,A 180.000,B 0.000,C 180.000} C_DIS
LIN {X 106.752,Y 109.304,Z 66.067,A 180.000,B 0.000,C 180.000} C_DIS
LIN {X 106.815,Y 109.257,Z 66.065,A 180.000,B 0.000,C 180.000} C_DIS
LIN {X 106.877,Y 109.208,Z 66.062,A 180.000,B 0.000,C 180.000} C_DIS
LIN {X 106.937,Y 109.157,Z 66.059,A 180.000,B 0.000,C 180.000} C_DIS
LIN {X 107.418,Y 108.751,Z 66.037,A 180.000,B 0.000,C 180.000} C_DIS
LIN {X 107.478,Y 108.700,Z 66.034,A 180.000,B 0.000,C 180.000} C_DIS
LIN {X 107.537,Y 108.647,Z 66.032,A 180.000,B 0.000,C 180.000} C_DIS
LIN {X 107.594,Y 108.593,Z 66.029,A 180.000,B 0.000,C 180.000} C_DIS
LIN {X 108.052,Y 108.160,Z 66.007,A 180.000,B 0.000,C 180.000} C_DIS
LIN {X 108.108,Y 108.105,Z 66.004,A 180.000,B 0.000,C 180.000} C_DIS
LIN {X 108.163,Y 108.048,Z 66.001,A 180.000,B 0.000,C 180.000} C_DIS
LIN {X 108.596,Y 107.591,Z 65.979,A 180.000,B 0.000,C 180.000} C_DIS
LIN {X 108.650,Y 107.533,Z 65.977,A 180.000,B 0.000,C 180.000} C_DIS
LIN {X 108.703,Y 107.475,Z 65.974,A 180.000,B 0.000,C 180.000} C_DIS
LIN {X 108.754,Y 107.415,Z 65.971,A 180.000,B 0.000,C 180.000} C_DIS
LIN {X 109.160,Y 106.934,Z 65.949,A 180.000,B 0.000,C 180.000} C_DIS
LIN {X 109.211,Y 106.873,Z 65.946,A 180.000,B 0.000,C 180.000} C_DIS
LIN {X 109.259,Y 106.811,Z 65.944,A 180.000,B 0.000,C 180.000} C_DIS
LIN {X 109.307,Y 106.748,Z 65.941,A 180.000,B 0.000,C 180.000} C_DIS
LIN {X 109.686,Y 106.245,Z 65.919,A 180.000,B 0.000,C 180.000} C_DIS
LIN {X 109.732,Y 106.182,Z 65.916,A 180.000,B 0.000,C 180.000} C_DIS
LIN {X 109.777,Y 106.117,Z 65.913,A 180.000,B 0.000,C 180.000} C_DIS
LIN {X 109.908,Y 105.920,Z 65.905,A 180.000,B 0.000,C 180.000} C_DIS
LIN {X 110.127,Y 105.593,Z 65.891,A 180.000,B 0.000,C 180.000} C_DIS
LIN {X 110.171,Y 105.527,Z 65.889,A 180.000,B 0.000,C 180.000} C_DIS
LIN {X 110.213,Y 105.461,Z 65.886,A 180.000,B 0.000,C 180.000} C_DIS
LIN {X 110.253,Y 105.393,Z 65.883,A 180.000,B 0.000,C 180.000} C_DIS
LIN {X 110.573,Y 104.851,Z 65.861,A 180.000,B 0.000,C 180.000} C_DIS
LIN {X 110.613,Y 104.783,Z 65.858,A 180.000,B 0.000,C 180.000} C_DIS
LIN {X 110.651,Y 104.714,Z 65.856,A 180.000,B 0.000,C 180.000} C_DIS
LIN {X 110.687,Y 104.644,Z 65.853,A 180.000,B 0.000,C 180.000} C_DIS
LIN {X 110.904,Y 104.224,Z 65.836,A 180.000,B 0.000,C 180.000} C_DIS
LIN {X 110.976,Y 104.084,Z 65.831,A 180.000,B 0.000,C 180.000} C_DIS
LIN {X 111.012,Y 104.014,Z 65.828,A 180.000,B 0.000,C 180.000} C_DIS
LIN {X 111.045,Y 103.942,Z 65.825,A 180.000,B 0.000,C 180.000} C_DIS
LIN {X 111.077,Y 103.870,Z 65.823,A 180.000,B 0.000,C 180.000} C_DIS
LIN {X 111.142,Y 103.727,Z 65.817,A 180.000,B 0.000,C 180.000} C_DIS
LIN {X 111.302,Y 103.367,Z 65.803,A 180.000,B 0.000,C 180.000} C_DIS
LIN {X 111.335,Y 103.295,Z 65.801,A 180.000,B 0.000,C 180.000} C_DIS
LIN {X 111.365,Y 103.223,Z 65.798,A 180.000,B 0.000,C 180.000} C_DIS
LIN {X 111.394,Y 103.149,Z 65.795,A 180.000,B 0.000,C 180.000} C_DIS
LIN {X 111.562,Y 102.708,Z 65.779,A 180.000,B 0.000,C 180.000} C_DIS
LIN {X 111.619,Y 102.561,Z 65.773,A 180.000,B 0.000,C 180.000} C_DIS
LIN {X 111.646,Y 102.487,Z 65.770,A 180.000,B 0.000,C 180.000} C_DIS
LIN {X 111.672,Y 102.413,Z 65.768,A 180.000,B 0.000,C 180.000} C_DIS
LIN {X 111.696,Y 102.338,Z 65.765,A 180.000,B 0.000,C 180.000} C_DIS
LIN {X 111.744,Y 102.188,Z 65.759,A 180.000,B 0.000,C 180.000} C_DIS
LIN {X 111.768,Y 102.113,Z 65.757,A 180.000,B 0.000,C 180.000} C_DIS
LIN {X 111.816,Y 101.963,Z 65.751,A 180.000,B 0.000,C 180.000} C_DIS
LIN {X 111.888,Y 101.738,Z 65.743,A 180.000,B 0.000,C 180.000} C_DIS
LIN {X 111.911,Y 101.662,Z 65.740,A 180.000,B 0.000,C 180.000} C_DIS
LIN {X 111.932,Y 101.586,Z 65.737,A 180.000,B 0.000,C 180.000} C_DIS
LIN {X 111.951,Y 101.510,Z 65.735,A 180.000,B 0.000,C 180.000} C_DIS
LIN {X 111.991,Y 101.358,Z 65.729,A 180.000,B 0.000,C 180.000} C_DIS
LIN {X 112.050,Y 101.129,Z 65.721,A 180.000,B 0.000,C 180.000} C_DIS
LIN {X 112.089,Y 100.976,Z 65.715,A 180.000,B 0.000,C 180.000} C_DIS
LIN {X 112.109,Y 100.900,Z 65.713,A 180.000,B 0.000,C 180.000} C_DIS
LIN {X 112.127,Y 100.824,Z 65.710,A 180.000,B 0.000,C 180.000} C_DIS
LIN {X 112.143,Y 100.746,Z 65.707,A 180.000,B 0.000,C 180.000} C_DIS
LIN {X 112.189,Y 100.515,Z 65.699,A 180.000,B 0.000,C 180.000} C_DIS
LIN {X 112.220,Y 100.360,Z 65.693,A 180.000,B 0.000,C 180.000} C_DIS
LIN {X 112.266,Y 100.129,Z 65.685,A 180.000,B 0.000,C 180.000} C_DIS
LIN {X 112.281,Y 100.051,Z 65.682,A 180.000,B 0.000,C 180.000} C_DIS
LIN {X 112.294,Y 99.974,Z 65.680,A 180.000,B 0.000,C 180.000} C_DIS
LIN {X 112.306,Y 99.896,Z 65.677,A 180.000,B 0.000,C 180.000} C_DIS
LIN {X 112.328,Y 99.740,Z 65.672,A 180.000,B 0.000,C 180.000} C_DIS
LIN {X 112.350,Y 99.584,Z 65.666,A 180.000,B 0.000,C 180.000} C_DIS
LIN {X 112.361,Y 99.506,Z 65.664,A 180.000,B 0.000,C 180.000} C_DIS
LIN {X 112.372,Y 99.428,Z 65.661,A 180.000,B 0.000,C 180.000} C_DIS
LIN {X 112.383,Y 99.350,Z 65.659,A 180.000,B 0.000,C 180.000} C_DIS
LIN {X 112.394,Y 99.272,Z 65.656,A 180.000,B 0.000,C 180.000} C_DIS
LIN {X 112.404,Y 99.194,Z 65.654,A 180.000,B 0.000,C 180.000} C_DIS
LIN {X 112.412,Y 99.115,Z 65.651,A 180.000,B 0.000,C 180.000} C_DIS
LIN {X 112.419,Y 99.037,Z 65.649,A 180.000,B 0.000,C 180.000} C_DIS
LIN {X 112.432,Y 98.880,Z 65.644,A 180.000,B 0.000,C 180.000} C_DIS
LIN {X 112.445,Y 98.723,Z 65.639,A 180.000,B 0.000,C 180.000} C_DIS
LIN {X 112.458,Y 98.566,Z 65.634,A 180.000,B 0.000,C 180.000} C_DIS
LIN {X 112.472,Y 98.409,Z 65.629,A 180.000,B 0.000,C 180.000} C_DIS
LIN {X 112.480,Y 98.252,Z 65.624,A 180.000,B 0.000,C 180.000} C_DIS
LIN {X 112.484,Y 98.095,Z 65.620,A 180.000,B 0.000,C 180.000} C_DIS
LIN {X 112.489,Y 97.937,Z 65.615,A 180.000,B 0.000,C 180.000} C_DIS
LIN {X 112.493,Y 97.780,Z 65.611,A 180.000,B 0.000,C 180.000} C_DIS
LIN {X 112.498,Y 97.622,Z 65.606,A 180.000,B 0.000,C 180.000} C_DIS
LIN {X 112.500,Y 97.465,Z 65.602,A 180.000,B 0.000,C 180.000} C_DIS
LIN {X 112.496,Y 97.307,Z 65.597,A 180.000,B 0.000,C 180.000} C_DIS
LIN {X 112.491,Y 97.150,Z 65.593,A 180.000,B 0.000,C 180.000} C_DIS
LIN {X 112.487,Y 96.992,Z 65.589,A 180.000,B 0.000,C 180.000} C_DIS
LIN {X 112.482,Y 96.835,Z 65.585,A 180.000,B 0.000,C 180.000} C_DIS
LIN {X 112.477,Y 96.678,Z 65.581,A 180.000,B 0.000,C 180.000} C_DIS
LIN {X 112.466,Y 96.520,Z 65.577,A 180.000,B 0.000,C 180.000} C_DIS
LIN {X 112.452,Y 96.364,Z 65.573,A 180.000,B 0.000,C 180.000} C_DIS
LIN {X 112.439,Y 96.207,Z 65.570,A 180.000,B 0.000,C 180.000} C_DIS
LIN {X 112.426,Y 96.050,Z 65.566,A 180.000,B 0.000,C 180.000} C_DIS
LIN {X 112.413,Y 95.893,Z 65.562,A 180.000,B 0.000,C 180.000} C_DIS
LIN {X 112.395,Y 95.736,Z 65.559,A 180.000,B 0.000,C 180.000} C_DIS
LIN {X 112.373,Y 95.580,Z 65.556,A 180.000,B 0.000,C 180.000} C_DIS
LIN {X 112.351,Y 95.424,Z 65.552,A 180.000,B 0.000,C 180.000} C_DIS
LIN {X 112.329,Y 95.268,Z 65.549,A 180.000,B 0.000,C 180.000} C_DIS
LIN {X 112.307,Y 95.112,Z 65.546,A 180.000,B 0.000,C 180.000} C_DIS
LIN {X 112.283,Y 94.957,Z 65.543,A 180.000,B 0.000,C 180.000} C_DIS
LIN {X 112.252,Y 94.802,Z 65.540,A 180.000,B 0.000,C 180.000} C_DIS
LIN {X 112.222,Y 94.648,Z 65.537,A 180.000,B 0.000,C 180.000} C_DIS
LIN {X 112.191,Y 94.493,Z 65.534,A 180.000,B 0.000,C 180.000} C_DIS
LIN {X 112.160,Y 94.339,Z 65.532,A 180.000,B 0.000,C 180.000} C_DIS
LIN {X 112.129,Y 94.184,Z 65.529,A 180.000,B 0.000,C 180.000} C_DIS
LIN {X 112.091,Y 94.031,Z 65.527,A 180.000,B 0.000,C 180.000} C_DIS
LIN {X 112.013,Y 93.726,Z 65.522,A 180.000,B 0.000,C 180.000} C_DIS
LIN {X 111.934,Y 93.421,Z 65.518,A 180.000,B 0.000,C 180.000} C_DIS
LIN {X 111.842,Y 93.120,Z 65.514,A 180.000,B 0.000,C 180.000} C_DIS
LIN {X 111.747,Y 92.820,Z 65.511,A 180.000,B 0.000,C 180.000} C_DIS
LIN {X 111.649,Y 92.520,Z 65.508,A 180.000,B 0.000,C 180.000} C_DIS
LIN {X 111.537,Y 92.226,Z 65.505,A 180.000,B 0.000,C 180.000} C_DIS
LIN {X 111.425,Y 91.932,Z 65.503,A 180.000,B 0.000,C 180.000} C_DIS
LIN {X 111.306,Y 91.640,Z 65.502,A 180.000,B 0.000,C 180.000} C_DIS
LIN {X 111.177,Y 91.353,Z 65.501,A 180.000,B 0.000,C 180.000} C_DIS
LIN {X 111.048,Y 91.065,Z 65.500,A 180.000,B 0.000,C 180.000} C_DIS
LIN {X 110.946,Y 90.857,Z 65.500,A 180.000,B 0.000,C 180.000} C_DIS
; Cutting Move Starts
LIN {X 110.926,Y 90.818,Z 65.500,A 180.000,B 0.000,C 180.000} C_DIS
LIN {X 110.662,Y 90.307,Z 65.500,A 180.000,B 0.000,C 180.000} C_DIS
LIN {X 110.649,Y 90.282,Z 65.500,A 180.000,B 0.000,C 180.000} C_DIS
LIN {X 110.546,Y 90.103,Z 65.500,A 180.000,B 0.000,C 180.000} C_DIS
LIN {X 110.304,Y 89.693,Z 65.500,A 180.000,B 0.000,C 180.000} C_DIS
LIN {X 110.230,Y 89.567,Z 65.500,A 180.000,B 0.000,C 180.000} C_DIS
LIN {X 110.126,Y 89.405,Z 65.500,A 180.000,B 0.000,C 180.000} C_DIS
LIN {X 109.875,Y 89.031,Z 65.500,A 180.000,B 0.000,C 180.000} C_DIS
LIN {X 109.768,Y 88.870,Z 65.500,A 180.000,B 0.000,C 180.000} C_DIS
LIN {X 109.756,Y 88.852,Z 65.500,A 180.000,B 0.000,C 180.000} C_DIS
LIN {X 109.624,Y 88.673,Z 65.500,A 180.000,B 0.000,C 180.000} C_DIS
LIN {X 109.355,Y 88.316,Z 65.500,A 180.000,B 0.000,C 180.000} C_DIS
LIN {X 109.232,Y 88.153,Z 65.500,A 180.000,B 0.000,C 180.000} C_DIS
LIN {X 109.219,Y 88.137,Z 65.500,A 180.000,B 0.000,C 180.000} C_DIS
LIN {X 109.069,Y 87.958,Z 65.500,A 180.000,B 0.000,C 180.000} C_DIS
LIN {X 108.767,Y 87.601,Z 65.500,A 180.000,B 0.000,C 180.000} C_DIS
LIN {X 108.695,Y 87.517,Z 65.500,A 180.000,B 0.000,C 180.000} C_DIS
LIN {X 108.607,Y 87.422,Z 65.500,A 180.000,B 0.000,C 180.000} C_DIS
LIN {X 108.159,Y 86.947,Z 65.500,A 180.000,B 0.000,C 180.000} C_DIS
LIN {X 108.099,Y 86.885,Z 65.500,A 180.000,B 0.000,C 180.000} C_DIS
LIN {X 107.980,Y 86.773,Z 65.500,A 180.000,B 0.000,C 180.000} C_DIS
LIN {X 107.623,Y 86.435,Z 65.500,A 180.000,B 0.000,C 180.000} C_DIS
LIN {X 107.532,Y 86.349,Z 65.500,A 180.000,B 0.000,C 180.000} C_DIS
LIN {X 107.444,Y 86.271,Z 65.500,A 180.000,B 0.000,C 180.000} C_DIS
LIN {X 106.908,Y 85.818,Z 65.500,A 180.000,B 0.000,C 180.000} C_DIS
LIN {X 106.902,Y 85.813,Z 65.500,A 180.000,B 0.000,C 180.000} C_DIS
LIN {X 106.729,Y 85.678,Z 65.500,A 180.000,B 0.000,C 180.000} C_DIS
LIN {X 106.371,Y 85.409,Z 65.500,A 180.000,B 0.000,C 180.000} C_DIS
LIN {X 106.194,Y 85.276,Z 65.500,A 180.000,B 0.000,C 180.000} C_DIS
LIN {X 106.193,Y 85.276,Z 65.500,A 180.000,B 0.000,C 180.000} C_DIS
LIN {X 106.014,Y 85.154,Z 65.500,A 180.000,B 0.000,C 180.000} C_DIS
LIN {X 105.656,Y 84.915,Z 65.500,A 180.000,B 0.000,C 180.000} C_DIS
LIN {X 105.477,Y 84.797,Z 65.500,A 180.000,B 0.000,C 180.000} C_DIS
LIN {X 105.382,Y 84.740,Z 65.500,A 180.000,B 0.000,C 180.000} C_DIS
LIN {X 104.941,Y 84.480,Z 65.500,A 180.000,B 0.000,C 180.000} C_DIS
LIN {X 104.775,Y 84.383,Z 65.500,A 180.000,B 0.000,C 180.000} C_DIS
LIN {X 104.762,Y 84.375,Z 65.500,A 180.000,B 0.000,C 180.000} C_DIS
LIN {X 104.584,Y 84.282,Z 65.500,A 180.000,B 0.000,C 180.000} C_DIS
LIN {X 104.087,Y 84.025,Z 65.500,A 180.000,B 0.000,C 180.000} C_DIS
LIN {X 104.047,Y 84.005,Z 65.500,A 180.000,B 0.000,C 180.000} C_DIS
LIN {X 103.869,Y 83.922,Z 65.500,A 180.000,B 0.000,C 180.000} C_DIS
LIN {X 103.300,Y 83.668,Z 65.500,A 180.000,B 0.000,C 180.000} C_DIS
LIN {X 103.153,Y 83.608,Z 65.500,A 180.000,B 0.000,C 180.000} C_DIS
LIN {X 102.617,Y 83.403,Z 65.500,A 180.000,B 0.000,C 180.000} C_DIS
LIN {X 102.438,Y 83.336,Z 65.500,A 180.000,B 0.000,C 180.000} C_DIS
LIN {X 102.358,Y 83.310,Z 65.500,A 180.000,B 0.000,C 180.000} C_DIS
LIN {X 101.723,Y 83.108,Z 65.500,A 180.000,B 0.000,C 180.000} C_DIS
LIN {X 101.545,Y 83.057,Z 65.500,A 180.000,B 0.000,C 180.000} C_DIS
LIN {X 101.008,Y 82.919,Z 65.500,A 180.000,B 0.000,C 180.000} C_DIS
LIN {X 100.829,Y 82.874,Z 65.500,A 180.000,B 0.000,C 180.000} C_DIS
LIN {X 100.651,Y 82.838,Z 65.500,A 180.000,B 0.000,C 180.000} C_DIS
LIN {X 100.114,Y 82.731,Z 65.500,A 180.000,B 0.000,C 180.000} C_DIS
LIN {X 99.936,Y 82.700,Z 65.500,A 180.000,B 0.000,C 180.000} C_DIS
LIN {X 99.399,Y 82.624,Z 65.500,A 180.000,B 0.000,C 180.000} C_DIS
LIN {X 99.221,Y 82.599,Z 65.500,A 180.000,B 0.000,C 180.000} C_DIS
LIN {X 99.185,Y 82.595,Z 65.500,A 180.000,B 0.000,C 180.000} C_DIS
LIN {X 99.042,Y 82.582,Z 65.500,A 180.000,B 0.000,C 180.000} C_DIS
LIN {X 98.505,Y 82.536,Z 65.500,A 180.000,B 0.000,C 180.000} C_DIS
LIN {X 98.327,Y 82.523,Z 65.500,A 180.000,B 0.000,C 180.000} C_DIS
LIN {X 98.148,Y 82.517,Z 65.500,A 180.000,B 0.000,C 180.000} C_DIS
LIN {X 97.612,Y 82.502,Z 65.500,A 180.000,B 0.000,C 180.000} C_DIS
LIN {X 97.433,Y 82.501,Z 65.500,A 180.000,B 0.000,C 180.000} C_DIS
LIN {X 96.897,Y 82.516,Z 65.500,A 180.000,B 0.000,C 180.000} C_DIS
LIN {X 96.718,Y 82.521,Z 65.500,A 180.000,B 0.000,C 180.000} C_DIS
LIN {X 96.539,Y 82.533,Z 65.500,A 180.000,B 0.000,C 180.000} C_DIS
LIN {X 96.003,Y 82.578,Z 65.500,A 180.000,B 0.000,C 180.000} C_DIS
LIN {X 95.824,Y 82.594,Z 65.500,A 180.000,B 0.000,C 180.000} C_DIS
LIN {X 95.815,Y 82.595,Z 65.500,A 180.000,B 0.000,C 180.000} C_DIS
LIN {X 95.645,Y 82.618,Z 65.500,A 180.000,B 0.000,C 180.000} C_DIS
LIN {X 95.109,Y 82.694,Z 65.500,A 180.000,B 0.000,C 180.000} C_DIS
LIN {X 94.930,Y 82.722,Z 65.500,A 180.000,B 0.000,C 180.000} C_DIS
LIN {X 94.751,Y 82.758,Z 65.500,A 180.000,B 0.000,C 180.000} C_DIS
LIN {X 94.394,Y 82.829,Z 65.500,A 180.000,B 0.000,C 180.000} C_DIS
LIN {X 94.215,Y 82.865,Z 65.500,A 180.000,B 0.000,C 180.000} C_DIS
LIN {X 94.036,Y 82.908,Z 65.500,A 180.000,B 0.000,C 180.000} C_DIS
LIN {X 93.500,Y 83.046,Z 65.500,A 180.000,B 0.000,C 180.000} C_DIS
LIN {X 93.321,Y 83.094,Z 65.500,A 180.000,B 0.000,C 180.000} C_DIS
LIN {X 93.203,Y 83.131,Z 65.500,A 180.000,B 0.000,C 180.000} C_DIS
LIN {X 92.642,Y 83.310,Z 65.500,A 180.000,B 0.000,C 180.000} C_DIS
LIN {X 92.606,Y 83.322,Z 65.500,A 180.000,B 0.000,C 180.000} C_DIS
LIN {X 92.427,Y 83.386,Z 65.500,A 180.000,B 0.000,C 180.000} C_DIS
LIN {X 91.891,Y 83.591,Z 65.500,A 180.000,B 0.000,C 180.000} C_DIS
LIN {X 91.712,Y 83.662,Z 65.500,A 180.000,B 0.000,C 180.000} C_DIS
LIN {X 91.700,Y 83.668,Z 65.500,A 180.000,B 0.000,C 180.000} C_DIS
LIN {X 91.176,Y 83.902,Z 65.500,A 180.000,B 0.000,C 180.000} C_DIS
LIN {X 90.997,Y 83.983,Z 65.500,A 180.000,B 0.000,C 180.000} C_DIS
LIN {X 90.913,Y 84.025,Z 65.500,A 180.000,B 0.000,C 180.000} C_DIS
LIN {X 90.461,Y 84.259,Z 65.500,A 180.000,B 0.000,C 180.000} C_DIS
LIN {X 90.282,Y 84.351,Z 65.500,A 180.000,B 0.000,C 180.000} C_DIS
LIN {X 90.225,Y 84.383,Z 65.500,A 180.000,B 0.000,C 180.000} C_DIS
LIN {X 90.103,Y 84.454,Z 65.500,A 180.000,B 0.000,C 180.000} C_DIS
LIN {X 89.618,Y 84.740,Z 65.500,A 180.000,B 0.000,C 180.000} C_DIS
LIN {X 89.567,Y 84.770,Z 65.500,A 180.000,B 0.000,C 180.000} C_DIS
LIN {X 89.388,Y 84.886,Z 65.500,A 180.000,B 0.000,C 180.000} C_DIS
LIN {X 89.031,Y 85.125,Z 65.500,A 180.000,B 0.000,C 180.000} C_DIS
LIN {X 88.852,Y 85.244,Z 65.500,A 180.000,B 0.000,C 180.000} C_DIS
LIN {X 88.806,Y 85.276,Z 65.500,A 180.000,B 0.000,C 180.000} C_DIS
LIN {X 88.673,Y 85.376,Z 65.500,A 180.000,B 0.000,C 180.000} C_DIS
LIN {X 88.316,Y 85.645,Z 65.500,A 180.000,B 0.000,C 180.000} C_DIS
LIN {X 88.137,Y 85.781,Z 65.500,A 180.000,B 0.000,C 180.000} C_DIS
LIN {X 88.098,Y 85.813,Z 65.500,A 180.000,B 0.000,C 180.000} C_DIS
